LIN {X 0,Y 114.701,Z 386.692,A -85,B 0,C 180,E1 -25992.159,E2 -25992.159} C_VEL
LIN {X 0,Y 112.816,Z 386.681,A -85,B 0,C 180,E1 -25999.228,E2 -25999.228} C_VEL
LIN {X 0,Y 112.467,Z 385.169,A -85,B 0,C 180,E1 -26006.417,E2 -26006.417} C_VEL
LIN {X 0,Y 112.641,Z 383.781,A -85,B 0,C 180,E1 -26009.999,E2 -26009.999} C_VEL
LIN {X 0,Y 112.455,Z 380.804,A -85,B 0,C 180,E1 -26015.378,E2 -26015.378} C_VEL
LIN {X 0,Y 112.837,Z 376.72,A -85,B 0,C 180,E1 -26020.769,E2 -26020.769} C_VEL
LIN {X 0,Y 114.222,Z 370.392,A -85,B 0,C 180,E1 -26026.993,E2 -26026.993} C_VEL
LIN {X 0,Y 116.442,Z 363.485,A -85,B 0,C 180,E1 -26032.161,E2 -26032.161} C_VEL
LIN {X 0,Y 118.813,Z 356.389,A -85,B 0,C 180,E1 -26036.336,E2 -26036.336} C_VEL
LIN {X 0,Y 120.686,Z 351.028,A -85,B 0,C 180,E1 -26038.937,E2 -26038.937} C_VEL
LIN {X 0,Y 123.681,Z 342.854,A -85,B 0,C 180,E1 -26042.189,E2 -26042.189} C_VEL
LIN {X 0,Y 127.076,Z 332.271,A -85,B 0,C 180,E1 -26045.5,E2 -26045.5} C_VEL
LIN {X 0,Y 129.058,Z 325.849,A -85,B 0,C 180,E1 -26047.105,E2 -26047.105} C_VEL
LIN {X 0,Y 129.821,Z 322.45,A -85,B 0,C 180,E1 -26047.931,E2 -26047.931} C_VEL
LIN {X 0,Y 129.907,Z 315.621,A -85,B 0,C 180,E1 -26049.725,E2 -26049.725} C_VEL
LIN {X 0,Y 129.031,Z 304.225,A -85,B 0,C 180,E1 -26052.426,E2 -26052.426} C_VEL
LIN {X 0,Y 129.487,Z 298.65,A -85,B 0,C 180,E1 -26053.261,E2 -26053.261} C_VEL
LIN {X 0,Y 129.674,Z 297.694,A -85,B 0,C 180,E1 -26053.354,E2 -26053.354} C_VEL
LIN {X 0,Y 131.69,Z 283.784,A -85,B 0,C 180,E1 -26054.55,E2 -26054.55} C_VEL
LIN {X 0,Y 134.432,Z 245.397,A -85,B 0,C 180,E1 -26056.42,E2 -26056.42} C_VEL
LIN {X 0,Y 133.527,Z 229.449,A -85,B 0,C 180,E1 -26057.848,E2 -26057.848} C_VEL
LIN {X 0,Y 129.833,Z 218.225,A -85,B 0,C 180,E1 -26060.042,E2 -26060.042} C_VEL
LIN {X 0,Y 125.815,Z 208.24,A -85,B 0,C 180,E1 -26062.464,E2 -26062.464} C_VEL
LIN {X 0,Y 123.844,Z 204.228,A -85,B 0,C 180,E1 -26063.668,E2 -26063.668} C_VEL
LIN {X 0,Y 119.247,Z 196.971,A -85,B 0,C 180,E1 -26066.553,E2 -26066.553} C_VEL
LIN {X 0,Y 116.624,Z 193.11,A -85,B 0,C 180,E1 -26068.355,E2 -26068.355} C_VEL
LIN {X 0,Y 114.457,Z 189.787,A -85,B 0,C 180,E1 -26069.974,E2 -26069.974} C_VEL
LIN {X 0,Y 112.098,Z 186.672,A -85,B 0,C 180,E1 -26071.824,E2 -26071.824} C_VEL
LIN {X 0,Y 111.318,Z 185.287,A -85,B 0,C 180,E1 -26072.504,E2 -26072.504} C_VEL
LIN {X 0,Y 109.012,Z 183.185,A -85,B 0,C 180,E1 -26074.399,E2 -26074.399} C_VEL
LIN {X 0,Y 107.991,Z 180.792,A -85,B 0,C 180,E1 -26075.47,E2 -26075.47} C_VEL
LIN {X 0,Y 107.875,Z 180.047,A -85,B 0,C 180,E1 -26075.795,E2 -26075.795} C_VEL
LIN {X 0,Y 107.882,Z 179.983,A -85,B 0,C 180,E1 -26080.99,E2 -26080.99} C_VEL
LIN {X 0,Y 108.226,Z 180,A -85,B 0,C 180,E1 -26088.765,E2 -26088.765} C_VEL
LIN {X 0,Y 108.441,Z 179.966,A -85,B 0,C 180,E1 -26096.283,E2 -26096.283} C_VEL
LIN {X 0,Y 108.917,Z 179.902,A -85,B 0,C 180,E1 -26099.999,E2 -26099.999} C_VEL
LIN {X 0,Y 108.304,Z 179.989,A -85,B 0,C 180,E1 -26107.456,E2 -26107.456} C_VEL
LIN {X 0,Y 108.174,Z 179.988,A -85,B 0,C 180,E1 -26112.96,E2 -26112.96} C_VEL
LIN {X 0,Y 107.903,Z 180.028,A -85,B 0,C 180,E1 -26119.005,E2 -26119.005} C_VEL
LIN {X 0,Y 107.855,Z 180.044,A -85,B 0,C 180,E1 -26124.182,E2 -26124.182} C_VEL
LIN {X 0,Y 107.778,Z 180.041,A -85,B 0,C 180,E1 -26132.039,E2 -26132.039} C_VEL
LIN {X 0,Y 107.688,Z 180.049,A -85,B 0,C 180,E1 -26138.451,E2 -26138.451} C_VEL
LIN {X 0,Y 107.687,Z 180.208,A -85,B 0,C 180,E1 -26144.963,E2 -26144.963} C_VEL
LIN {X 0,Y 108.581,Z 182.753,A -85,B 0,C 180,E1 -26145.968,E2 -26145.968} C_VEL
LIN {X 0,Y 110.766,Z 185.022,A -85,B 0,C 180,E1 -26147.829,E2 -26147.829} C_VEL
LIN {X 0,Y 111.609,Z 185.761,A -85,B 0,C 180,E1 -26148.498,E2 -26148.498} C_VEL
LIN {X 0,Y 113.569,Z 188.992,A -85,B 0,C 180,E1 -26150.138,E2 -26150.138} C_VEL
LIN {X 0,Y 115.129,Z 190.684,A -85,B 0,C 180,E1 -26151.28,E2 -26151.28} C_VEL
LIN {X 0,Y 120.859,Z 199.285,A -85,B 0,C 180,E1 -26155.238,E2 -26155.238} C_VEL
LIN {X 0,Y 125.031,Z 206.174,A -85,B 0,C 180,E1 -26157.785,E2 -26157.785} C_VEL
LIN {X 0,Y 130.851,Z 217.027,A -85,B 0,C 180,E1 -26161.01,E2 -26161.01} C_VEL
LIN {X 0,Y 135.488,Z 227.713,A -85,B 0,C 180,E1 -26163.46,E2 -26163.46} C_VEL
LIN {X 0,Y 132.145,Z 273.455,A -85,B 0,C 180,E1 -26165.609,E2 -26165.609} C_VEL
LIN {X 0,Y 130.472,Z 286.832,A -85,B 0,C 180,E1 -26166.792,E2 -26166.792} C_VEL
LIN {X 0,Y 128.112,Z 299.797,A -85,B 0,C 180,E1 -26168.525,E2 -26168.525} C_VEL
LIN {X 0,Y 125.177,Z 311.686,A -85,B 0,C 180,E1 -26170.741,E2 -26170.741} C_VEL
LIN {X 0,Y 121.73,Z 323.3,A -85,B 0,C 180,E1 -26173.654,E2 -26173.654} C_VEL
LIN {X 0,Y 118.203,Z 333.75,A -85,B 0,C 180,E1 -26177.118,E2 -26177.118} C_VEL
LIN {X 0,Y 114.672,Z 343.135,A -85,B 0,C 180,E1 -26181.187,E2 -26181.187} C_VEL
LIN {X 0,Y 111.181,Z 352.262,A -85,B 0,C 180,E1 -26186.376,E2 -26186.376} C_VEL
LIN {X 0,Y 108.53,Z 359.552,A -85,B 0,C 180,E1 -26191.856,E2 -26191.856} C_VEL
LIN {X 0,Y 106.453,Z 365.739,A -85,B 0,C 180,E1 -26197.993,E2 -26197.993} C_VEL
LIN {X 0,Y 105.375,Z 369.965,A -85,B 0,C 180,E1 -26203.5,E2 -26203.5} C_VEL
LIN {X 0,Y 104.938,Z 373.8,A -85,B 0,C 180,E1 -26210.347,E2 -26210.347} C_VEL
LIN {X 0,Y 105.788,Z 376.41,A -85,B 0,C 180,E1 -26217.714,E2 -26217.714} C_VEL
LIN {X 0,Y 106.874,Z 377.199,A -85,B 0,C 180,E1 -26221.742,E2 -26221.742} C_VEL
LIN {X 0,Y 108.366,Z 377.569,A -85,B 0,C 180,E1 -26225.711,E2 -26225.711} C_VEL
LIN {X 0,Y 110.875,Z 377.373,A -85,B 0,C 180,E1 -26230.48,E2 -26230.48} C_VEL
LIN {X 0,Y 115.497,Z 375.922,A -85,B 0,C 180,E1 -26236.904,E2 -26236.904} C_VEL
LIN {X 0,Y 118.712,Z 374.445,A -85,B 0,C 180,E1 -26240.321,E2 -26240.321} C_VEL
LIN {X 0,Y 125.327,Z 370.597,A -85,B 0,C 180,E1 -26245.891,E2 -26245.891} C_VEL
LIN {X 0,Y 132.858,Z 365.177,A -85,B 0,C 180,E1 -26250.79,E2 -26250.79} C_VEL
LIN {X 0,Y 140.026,Z 358.919,A -85,B 0,C 180,E1 -26254.614,E2 -26254.614} C_VEL
LIN {X 0,Y 147.752,Z 351.022,A -85,B 0,C 180,E1 -26258.03,E2 -26258.03} C_VEL
LIN {X 0,Y 154.642,Z 342.793,A -85,B 0,C 180,E1 -26260.567,E2 -26260.567} C_VEL
LIN {X 0,Y 161.719,Z 332.547,A -85,B 0,C 180,E1 -26262.957,E2 -26262.957} C_VEL
LIN {X 0,Y 167.578,Z 322.406,A -85,B 0,C 180,E1 -26264.709,E2 -26264.709} C_VEL
LIN {X 0,Y 172.609,Z 311.679,A -85,B 0,C 180,E1 -26266.157,E2 -26266.157} C_VEL
LIN {X 0,Y 176.952,Z 300.005,A -85,B 0,C 180,E1 -26267.306,E2 -26267.306} C_VEL
LIN {X 0,Y 180.318,Z 287.878,A -85,B 0,C 180,E1 -26268.188,E2 -26268.188} C_VEL
LIN {X 0,Y 182.718,Z 275.29,A -85,B 0,C 180,E1 -26268.804,E2 -26268.804} C_VEL
LIN {X 0,Y 183.684,Z 266.817,A -85,B 0,C 180,E1 -26269.111,E2 -26269.111} C_VEL
LIN {X 0,Y 180.644,Z 260.298,A -85,B 0,C 180,E1 -26272.521,E2 -26272.521} C_VEL
LIN {X 0,Y 177.733,Z 254.302,A -85,B 0,C 180,E1 -26276.657,E2 -26276.657} C_VEL
LIN {X 0,Y 176.128,Z 251.308,A -85,B 0,C 180,E1 -26279.593,E2 -26279.593} C_VEL
LIN {X 0,Y 174.589,Z 248.05,A -85,B 0,C 180,E1 -26284.04,E2 -26284.04} C_VEL
LIN {X 0,Y 174.347,Z 247.326,A -85,B 0,C 180,E1 -26285.204,E2 -26285.204} C_VEL
LIN {X 0,Y 173.89,Z 247.213,A -85,B 0,C 180,E1 -26291.659,E2 -26291.659} C_VEL
LIN {X 0,Y 174.227,Z 247.599,A -85,B 0,C 180,E1 -26293.856,E2 -26293.856} C_VEL
LIN {X 0,Y 175.605,Z 251.412,A -85,B 0,C 180,E1 -26298.89,E2 -26298.89} C_VEL
LIN {X 0,Y 176.463,Z 253.601,A -85,B 0,C 180,E1 -26300.831,E2 -26300.831} C_VEL
LIN {X 0,Y 178.028,Z 257.372,A -85,B 0,C 180,E1 -26303.634,E2 -26303.634} C_VEL
LIN {X 0,Y 179.981,Z 262.71,A -85,B 0,C 180,E1 -26306.563,E2 -26306.563} C_VEL
LIN {X 0,Y 182.016,Z 268.722,A -85,B 0,C 180,E1 -26309.175,E2 -26309.175} C_VEL
LIN {X 0,Y 183.184,Z 272.321,A -85,B 0,C 180,E1 -26310.497,E2 -26310.497} C_VEL
LIN {X 0,Y 181.43,Z 286.139,A -85,B 0,C 180,E1 -26311.025,E2 -26311.025} C_VEL
LIN {X 0,Y 178.365,Z 299.021,A -85,B 0,C 180,E1 -26311.617,E2 -26311.617} C_VEL
LIN {X 0,Y 174.048,Z 312.047,A -85,B 0,C 180,E1 -26312.549,E2 -26312.549} C_VEL
LIN {X 0,Y 168.989,Z 323.707,A -85,B 0,C 180,E1 -26313.718,E2 -26313.718} C_VEL
LIN {X 0,Y 162.609,Z 335.397,A -85,B 0,C 180,E1 -26315.335,E2 -26315.335} C_VEL
LIN {X 0,Y 156.424,Z 344.847,A -85,B 0,C 180,E1 -26317.108,E2 -26317.108} C_VEL
LIN {X 0,Y 149.851,Z 353.495,A -85,B 0,C 180,E1 -26319.299,E2 -26319.299} C_VEL
LIN {X 0,Y 142.285,Z 361.956,A -85,B 0,C 180,E1 -26322.191,E2 -26322.191} C_VEL
LIN {X 0,Y 135.158,Z 368.785,A -85,B 0,C 180,E1 -26325.413,E2 -26325.413} C_VEL
LIN {X 0,Y 128.542,Z 374.292,A -85,B 0,C 180,E1 -26328.997,E2 -26328.997} C_VEL
LIN {X 0,Y 121.331,Z 379.649,A -85,B 0,C 180,E1 -26334.189,E2 -26334.189} C_VEL
LIN {X 0,Y 117.646,Z 381.979,A -85,B 0,C 180,E1 -26337.476,E2 -26337.476} C_VEL
LIN {X 0,Y 111.974,Z 384.967,A -85,B 0,C 180,E1 -26343.937,E2 -26343.937} C_VEL
LIN {X 0,Y 109.699,Z 385.885,A -85,B 0,C 180,E1 -26347.393,E2 -26347.393} C_VEL
LIN {X 0,Y 106.683,Z 386.525,A -85,B 0,C 180,E1 -26354.721,E2 -26354.721} C_VEL
LIN {X 0,Y 105.409,Z 385.676,A -85,B 0,C 180,E1 -26362.336,E2 -26362.336} C_VEL
LIN {X 0,Y 105.48,Z 383.981,A -85,B 0,C 180,E1 -26368.092,E2 -26368.092} C_VEL
LIN {X 0,Y 105.459,Z 382.498,A -85,B 0,C 180,E1 -26371.524,E2 -26371.524} C_VEL
LIN {X 0,Y 105.446,Z 378.874,A -85,B 0,C 180,E1 -26377.66,E2 -26377.66} C_VEL
LIN {X 0,Y 106.167,Z 374.293,A -85,B 0,C 180,E1 -26383.396,E2 -26383.396} C_VEL
LIN {X 0,Y 108.144,Z 367.298,A -85,B 0,C 180,E1 -26389.948,E2 -26389.948} C_VEL
LIN {X 0,Y 110.77,Z 359.68,A -85,B 0,C 180,E1 -26395.357,E2 -26395.357} C_VEL
LIN {X 0,Y 113.549,Z 351.859,A -85,B 0,C 180,E1 -26399.679,E2 -26399.679} C_VEL
LIN {X 0,Y 116.939,Z 343.453,A -85,B 0,C 180,E1 -26403.257,E2 -26403.257} C_VEL
LIN {X 0,Y 120.499,Z 333.091,A -85,B 0,C 180,E1 -26406.713,E2 -26406.713} C_VEL
LIN {X 0,Y 123.614,Z 323.202,A -85,B 0,C 180,E1 -26409.234,E2 -26409.234} C_VEL
LIN {X 0,Y 126.699,Z 311.658,A -85,B 0,C 180,E1 -26411.465,E2 -26411.465} C_VEL
LIN {X 0,Y 129.288,Z 300.08,A -85,B 0,C 180,E1 -26413.069,E2 -26413.069} C_VEL
LIN {X 0,Y 129.674,Z 297.694,A -85,B 0,C 180,E1 -26413.354,E2 -26413.354} C_VEL
LIN {X 0,Y 130.345,Z 292.966,A -85,B 0,C 180,E1 -26413.874,E2 -26413.874} C_VEL
LIN {X 0,Y 130.243,Z 290.151,A -85,B 0,C 180,E1 -26414.275,E2 -26414.275} C_VEL
LIN {X 0,Y 129.287,Z 282.732,A -85,B 0,C 180,E1 -26415.44,E2 -26415.44} C_VEL
LIN {X 0,Y 127.603,Z 273.348,A -85,B 0,C 180,E1 -26416.792,E2 -26416.792} C_VEL
LIN {X 0,Y 127.324,Z 267.511,A -85,B 0,C 180,E1 -26417.311,E2 -26417.311} C_VEL
LIN {X 0,Y 128.86,Z 244.337,A -85,B 0,C 180,E1 -26418.461,E2 -26418.461} C_VEL
LIN {X 0,Y 128.067,Z 231.4,A -85,B 0,C 180,E1 -26419.737,E2 -26419.737} C_VEL
LIN {X 0,Y 124.718,Z 220.97,A -85,B 0,C 180,E1 -26421.914,E2 -26421.914} C_VEL
LIN {X 0,Y 120.764,Z 211.039,A -85,B 0,C 180,E1 -26424.538,E2 -26424.538} C_VEL
LIN {X 0,Y 117.152,Z 204.663,A -85,B 0,C 180,E1 -26426.962,E2 -26426.962} C_VEL
LIN {X 0,Y 113.319,Z 198.721,A -85,B 0,C 180,E1 -26429.763,E2 -26429.763} C_VEL
LIN {X 0,Y 110.992,Z 195.236,A -85,B 0,C 180,E1 -26431.638,E2 -26431.638} C_VEL
LIN {X 0,Y 108.042,Z 191.063,A -85,B 0,C 180,E1 -26434.213,E2 -26434.213} C_VEL
LIN {X 0,Y 105.846,Z 188.492,A -85,B 0,C 180,E1 -26436.262,E2 -26436.262} C_VEL
LIN {X 0,Y 104.885,Z 186.451,A -85,B 0,C 180,E1 -26437.338,E2 -26437.338} C_VEL
LIN {X 0,Y 102.468,Z 184.637,A -85,B 0,C 180,E1 -26439.812,E2 -26439.812} C_VEL
LIN {X 0,Y 101.07,Z 182.025,A -85,B 0,C 180,E1 -26441.633,E2 -26441.633} C_VEL
LIN {X 0,Y 100.815,Z 180.859,A -85,B 0,C 180,E1 -26442.242,E2 -26442.242} C_VEL
LIN {X 0,Y 101.125,Z 180.879,A -85,B 0,C 180,E1 -26447.965,E2 -26447.965} C_VEL
LIN {X 0,Y 101.232,Z 180.856,A -85,B 0,C 180,E1 -26452.018,E2 -26452.018} C_VEL
LIN {X 0,Y 101.844,Z 180.782,A -85,B 0,C 180,E1 -26459.999,E2 -26459.999} C_VEL
LIN {X 0,Y 101.243,Z 180.866,A -85,B 0,C 180,E1 -26467.98,E2 -26467.98} C_VEL
LIN {X 0,Y 101.103,Z 180.87,A -85,B 0,C 180,E1 -26473.302,E2 -26473.302} C_VEL
LIN {X 0,Y 100.815,Z 180.902,A -85,B 0,C 180,E1 -26480.398,E2 -26480.398} C_VEL
LIN {X 0,Y 100.773,Z 180.93,A -85,B 0,C 180,E1 -26484.958,E2 -26484.958} C_VEL
LIN {X 0,Y 100.687,Z 180.932,A -85,B 0,C 180,E1 -26493.114,E2 -26493.114} C_VEL
LIN {X 0,Y 100.666,Z 180.974,A -85,B 0,C 180,E1 -26498.526,E2 -26498.526} C_VEL
LIN {X 0,Y 101.319,Z 183.24,A -85,B 0,C 180,E1 -26499.581,E2 -26499.581} C_VEL
LIN {X 0,Y 103.297,Z 185.672,A -85,B 0,C 180,E1 -26501.894,E2 -26501.894} C_VEL
LIN {X 0,Y 104.844,Z 186.814,A -85,B 0,C 180,E1 -26503.443,E2 -26503.443} C_VEL
LIN {X 0,Y 106.693,Z 189.893,A -85,B 0,C 180,E1 -26505.367,E2 -26505.367} C_VEL
LIN {X 0,Y 108.713,Z 192.013,A -85,B 0,C 180,E1 -26507.153,E2 -26507.153} C_VEL
LIN {X 0,Y 111.364,Z 195.716,A -85,B 0,C 180,E1 -26509.413,E2 -26509.413} C_VEL
LIN {X 0,Y 115.239,Z 201.557,A -85,B 0,C 180,E1 -26512.421,E2 -26512.421} C_VEL
LIN {X 0,Y 120.179,Z 209.544,A -85,B 0,C 180,E1 -26515.801,E2 -26515.801} C_VEL
LIN {X 0,Y 126.22,Z 221.191,A -85,B 0,C 180,E1 -26519.494,E2 -26519.494} C_VEL
LIN {X 0,Y 129.832,Z 229.561,A -85,B 0,C 180,E1 -26521.553,E2 -26521.553} C_VEL
LIN {X 0,Y 126.447,Z 274.354,A -85,B 0,C 180,E1 -26523.746,E2 -26523.746} C_VEL
LIN {X 0,Y 124.618,Z 287.912,A -85,B 0,C 180,E1 -26524.995,E2 -26524.995} C_VEL
LIN {X 0,Y 122.241,Z 300.262,A -85,B 0,C 180,E1 -26526.718,E2 -26526.718} C_VEL
LIN {X 0,Y 119.343,Z 311.486,A -85,B 0,C 180,E1 -26528.858,E2 -26528.858} C_VEL
LIN {X 0,Y 115.681,Z 323.201,A -85,B 0,C 180,E1 -26531.859,E2 -26531.859} C_VEL
LIN {X 0,Y 111.932,Z 333.741,A -85,B 0,C 180,E1 -26535.455,E2 -26535.455} C_VEL
LIN {X 0,Y 108.271,Z 343.007,A -85,B 0,C 180,E1 -26539.616,E2 -26539.616} C_VEL
LIN {X 0,Y 104.458,Z 352.362,A -85,B 0,C 180,E1 -26545.176,E2 -26545.176} C_VEL
LIN {X 0,Y 101.627,Z 359.708,A -85,B 0,C 180,E1 -26550.991,E2 -26550.991} C_VEL
LIN {X 0,Y 99.326,Z 366.195,A -85,B 0,C 180,E1 -26557.867,E2 -26557.867} C_VEL
LIN {X 0,Y 98.132,Z 370.85,A -85,B 0,C 180,E1 -26564.518,E2 -26564.518} C_VEL
LIN {X 0,Y 97.852,Z 374.164,A -85,B 0,C 180,E1 -26571.047,E2 -26571.047} C_VEL
LIN {X 0,Y 98.244,Z 375.791,A -85,B 0,C 180,E1 -26575.419,E2 -26575.419} C_VEL
LIN {X 0,Y 99.896,Z 377.43,A -85,B 0,C 180,E1 -26582.411,E2 -26582.411} C_VEL
LIN {X 0,Y 102.222,Z 377.932,A -85,B 0,C 180,E1 -26588.227,E2 -26588.227} C_VEL
LIN {X 0,Y 104.541,Z 377.719,A -85,B 0,C 180,E1 -26592.312,E2 -26592.312} C_VEL
LIN {X 0,Y 107.212,Z 377.092,A -85,B 0,C 180,E1 -26596.145,E2 -26596.145} C_VEL
LIN {X 0,Y 111.36,Z 375.573,A -85,B 0,C 180,E1 -26600.869,E2 -26600.869} C_VEL
LIN {X 0,Y 117.901,Z 372.339,A -85,B 0,C 180,E1 -26606.568,E2 -26606.568} C_VEL
LIN {X 0,Y 124.496,Z 368.233,A -85,B 0,C 180,E1 -26611.046,E2 -26611.046} C_VEL
LIN {X 0,Y 131.763,Z 362.775,A -85,B 0,C 180,E1 -26615.061,E2 -26615.061} C_VEL
LIN {X 0,Y 139.582,Z 355.769,A -85,B 0,C 180,E1 -26618.668,E2 -26618.668} C_VEL
LIN {X 0,Y 146.374,Z 348.696,A -85,B 0,C 180,E1 -26621.277,E2 -26621.277} C_VEL
LIN {X 0,Y 153.726,Z 339.698,A -85,B 0,C 180,E1 -26623.756,E2 -26623.756} C_VEL
LIN {X 0,Y 160.409,Z 329.813,A -85,B 0,C 180,E1 -26625.782,E2 -26625.782} C_VEL
LIN {X 0,Y 166.392,Z 319.026,A -85,B 0,C 180,E1 -26627.46,E2 -26627.46} C_VEL
LIN {X 0,Y 171.325,Z 308.107,A -85,B 0,C 180,E1 -26628.732,E2 -26628.732} C_VEL
LIN {X 0,Y 175.544,Z 296.066,A -85,B 0,C 180,E1 -26629.785,E2 -26629.785} C_VEL
LIN {X 0,Y 178.732,Z 283.464,A -85,B 0,C 180,E1 -26630.542,E2 -26630.542} C_VEL
LIN {X 0,Y 180.761,Z 270.84,A -85,B 0,C 180,E1 -26631.053,E2 -26631.053} C_VEL
LIN {X 0,Y 178.005,Z 264.538,A -85,B 0,C 180,E1 -26634.689,E2 -26634.689} C_VEL
LIN {X 0,Y 175.873,Z 260.138,A -85,B 0,C 180,E1 -26638.171,E2 -26638.171} C_VEL
LIN {X 0,Y 174.892,Z 258.049,A -85,B 0,C 180,E1 -26640.253,E2 -26640.253} C_VEL
LIN {X 0,Y 173.536,Z 254.812,A -85,B 0,C 180,E1 -26644.646,E2 -26644.646} C_VEL
LIN {X 0,Y 173.3,Z 254.338,A -85,B 0,C 180,E1 -26645.819,E2 -26645.819} C_VEL
LIN {X 0,Y 172.996,Z 254.247,A -85,B 0,C 180,E1 -26651.72,E2 -26651.72} C_VEL
LIN {X 0,Y 173.246,Z 254.591,A -85,B 0,C 180,E1 -26653.481,E2 -26653.481} C_VEL
LIN {X 0,Y 174.536,Z 258.424,A -85,B 0,C 180,E1 -26658.572,E2 -26658.572} C_VEL
LIN {X 0,Y 176.437,Z 263.611,A -85,B 0,C 180,E1 -26662.66,E2 -26662.66} C_VEL
LIN {X 0,Y 178.367,Z 269.331,A -85,B 0,C 180,E1 -26665.819,E2 -26665.819} C_VEL
LIN {X 0,Y 180.311,Z 275.713,A -85,B 0,C 180,E1 -26668.541,E2 -26668.541} C_VEL
LIN {X 0,Y 178.03,Z 289.665,A -85,B 0,C 180,E1 -26669.063,E2 -26669.063} C_VEL
LIN {X 0,Y 174.813,Z 301.773,A -85,B 0,C 180,E1 -26669.672,E2 -26669.672} C_VEL
LIN {X 0,Y 170.378,Z 313.955,A -85,B 0,C 180,E1 -26670.561,E2 -26670.561} C_VEL
LIN {X 0,Y 165.187,Z 325.092,A -85,B 0,C 180,E1 -26671.688,E2 -26671.688} C_VEL
LIN {X 0,Y 158.639,Z 336.483,A -85,B 0,C 180,E1 -26673.259,E2 -26673.259} C_VEL
LIN {X 0,Y 152.276,Z 345.689,A -85,B 0,C 180,E1 -26674.993,E2 -26674.993} C_VEL
LIN {X 0,Y 144.142,Z 355.597,A -85,B 0,C 180,E1 -26677.597,E2 -26677.597} C_VEL
LIN {X 0,Y 136.371,Z 363.605,A -85,B 0,C 180,E1 -26680.522,E2 -26680.522} C_VEL
LIN {X 0,Y 130.207,Z 369.07,A -85,B 0,C 180,E1 -26683.224,E2 -26683.224} C_VEL
LIN {X 0,Y 123.284,Z 374.455,A -85,B 0,C 180,E1 -26686.836,E2 -26686.836} C_VEL
LIN {X 0,Y 117.128,Z 378.697,A -85,B 0,C 180,E1 -26690.947,E2 -26690.947} C_VEL
LIN {X 0,Y 111.704,Z 381.924,A -85,B 0,C 180,E1 -26695.51,E2 -26695.51} C_VEL
LIN {X 0,Y 105.618,Z 384.809,A -85,B 0,C 180,E1 -26702.238,E2 -26702.238} C_VEL
LIN {X 0,Y 101.203,Z 386.087,A -85,B 0,C 180,E1 -26709.682,E2 -26709.682} C_VEL
LIN {X 0,Y 98.863,Z 385.891,A -85,B 0,C 180,E1 -26717.685,E2 -26717.685} C_VEL
LIN {X 0,Y 98.355,Z 385.224,A -85,B 0,C 180,E1 -26721.783,E2 -26721.783} C_VEL
LIN {X 0,Y 98.431,Z 383.287,A -85,B 0,C 180,E1 -26728.416,E2 -26728.416} C_VEL
LIN {X 0,Y 98.31,Z 380.639,A -85,B 0,C 180,E1 -26734.099,E2 -26734.099} C_VEL
LIN {X 0,Y 98.572,Z 376.721,A -85,B 0,C 180,E1 -26740.267,E2 -26740.267} C_VEL
LIN {X 0,Y 99.993,Z 370.632,A -85,B 0,C 180,E1 -26747.379,E2 -26747.379} C_VEL
LIN {X 0,Y 102.36,Z 363.924,A -85,B 0,C 180,E1 -26753.252,E2 -26753.252} C_VEL
LIN {X 0,Y 105.496,Z 355.533,A -85,B 0,C 180,E1 -26758.88,E2 -26758.88} C_VEL
LIN {X 0,Y 108.199,Z 348.95,A -85,B 0,C 180,E1 -26762.293,E2 -26762.293} C_VEL
LIN {X 0,Y 111.777,Z 339.734,A -85,B 0,C 180,E1 -26766.118,E2 -26766.118} C_VEL
LIN {X 0,Y 114.775,Z 331.263,A -85,B 0,C 180,E1 -26768.875,E2 -26768.875} C_VEL
LIN {X 0,Y 118.643,Z 319.446,A -85,B 0,C 180,E1 -26771.79,E2 -26771.79} C_VEL
LIN {X 0,Y 121.992,Z 306.784,A -85,B 0,C 180,E1 -26774.02,E2 -26774.02} C_VEL
LIN {X 0,Y 124.677,Z 293.418,A -85,B 0,C 180,E1 -26775.658,E2 -26775.658} C_VEL
LIN {X 0,Y 126.416,Z 280.076,A -85,B 0,C 180,E1 -26776.667,E2 -26776.667} C_VEL
LIN {X 0,Y 127.324,Z 267.511,A -85,B 0,C 180,E1 -26777.311,E2 -26777.311} C_VEL
LIN {X 0,Y 127.146,Z 261.686,A -85,B 0,C 180,E1 -26777.809,E2 -26777.809} C_VEL
LIN {X 0,Y 125.583,Z 252.305,A -85,B 0,C 180,E1 -26779.114,E2 -26779.114} C_VEL
LIN {X 0,Y 123.455,Z 241.084,A -85,B 0,C 180,E1 -26780.84,E2 -26780.84} C_VEL
LIN {X 0,Y 123.097,Z 237.226,A -85,B 0,C 180,E1 -26781.299,E2 -26781.299} C_VEL
LIN {X 0,Y 122.759,Z 233.368,A -85,B 0,C 180,E1 -26781.755,E2 -26781.755} C_VEL
LIN {X 0,Y 119.133,Z 222.078,A -85,B 0,C 180,E1 -26784.369,E2 -26784.369} C_VEL
LIN {X 0,Y 115.868,Z 214.01,A -85,B 0,C 180,E1 -26786.783,E2 -26786.783} C_VEL
LIN {X 0,Y 110.547,Z 204.935,A -85,B 0,C 180,E1 -26790.885,E2 -26790.885} C_VEL
LIN {X 0,Y 107.505,Z 200.444,A -85,B 0,C 180,E1 -26793.524,E2 -26793.524} C_VEL
LIN {X 0,Y 105.228,Z 197.043,A -85,B 0,C 180,E1 -26795.688,E2 -26795.688} C_VEL
LIN {X 0,Y 102.784,Z 193.818,A -85,B 0,C 180,E1 -26798.216,E2 -26798.216} C_VEL
LIN {X 0,Y 102.037,Z 192.616,A -85,B 0,C 180,E1 -26799.083,E2 -26799.083} C_VEL
LIN {X 0,Y 99.562,Z 190.02,A -85,B 0,C 180,E1 -26802.011,E2 -26802.011} C_VEL
LIN {X 0,Y 98.284,Z 187.472,A -85,B 0,C 180,E1 -26803.913,E2 -26803.913} C_VEL
LIN {X 0,Y 95.817,Z 185.626,A -85,B 0,C 180,E1 -26807.557,E2 -26807.557} C_VEL
LIN {X 0,Y 94.45,Z 183.265,A -85,B 0,C 180,E1 -26810.226,E2 -26810.226} C_VEL
LIN {X 0,Y 94.14,Z 181.743,A -85,B 0,C 180,E1 -26811.277,E2 -26811.277} C_VEL
LIN {X 0,Y 94.773,Z 181.661,A -85,B 0,C 180,E1 -26819.999,E2 -26819.999} C_VEL
LIN {X 0,Y 94.176,Z 181.741,A -85,B 0,C 180,E1 -26828.583,E2 -26828.583} C_VEL
LIN {X 0,Y 94.023,Z 181.753,A -85,B 0,C 180,E1 -26833.662,E2 -26833.662} C_VEL
LIN {X 0,Y 93.69,Z 181.789,A -85,B 0,C 180,E1 -26842.027,E2 -26842.027} C_VEL
LIN {X 0,Y 93.629,Z 181.964,A -85,B 0,C 180,E1 -26848.741,E2 -26848.741} C_VEL
LIN {X 0,Y 94.38,Z 184.288,A -85,B 0,C 180,E1 -26850.637,E2 -26850.637} C_VEL
LIN {X 0,Y 96.689,Z 186.837,A -85,B 0,C 180,E1 -26854.673,E2 -26854.673} C_VEL
LIN {X 0,Y 98.31,Z 187.833,A -85,B 0,C 180,E1 -26856.937,E2 -26856.937} C_VEL
LIN {X 0,Y 99.925,Z 190.819,A -85,B 0,C 180,E1 -26859.27,E2 -26859.27} C_VEL
LIN {X 0,Y 102.339,Z 193.289,A -85,B 0,C 180,E1 -26862.061,E2 -26862.061} C_VEL
LIN {X 0,Y 104.697,Z 196.675,A -85,B 0,C 180,E1 -26864.594,E2 -26864.594} C_VEL
LIN {X 0,Y 105.935,Z 198.189,A -85,B 0,C 180,E1 -26865.783,E2 -26865.783} C_VEL
LIN {X 0,Y 110.851,Z 205.318,A -85,B 0,C 180,E1 -26870.103,E2 -26870.103} C_VEL
LIN {X 0,Y 116.343,Z 214.711,A -85,B 0,C 180,E1 -26874.292,E2 -26874.292} C_VEL
LIN {X 0,Y 121.605,Z 225.166,A -85,B 0,C 180,E1 -26877.816,E2 -26877.816} C_VEL
LIN {X 0,Y 124.353,Z 231.71,A -85,B 0,C 180,E1 -26879.549,E2 -26879.549} C_VEL
LIN {X 0,Y 120.907,Z 274.78,A -85,B 0,C 180,E1 -26881.694,E2 -26881.694} C_VEL
LIN {X 0,Y 118.916,Z 288.704,A -85,B 0,C 180,E1 -26883.016,E2 -26883.016} C_VEL
LIN {X 0,Y 116.547,Z 300.366,A -85,B 0,C 180,E1 -26884.692,E2 -26884.692} C_VEL
LIN {X 0,Y 113.159,Z 312.786,A -85,B 0,C 180,E1 -26887.16,E2 -26887.16} C_VEL
LIN {X 0,Y 109.304,Z 324.329,A -85,B 0,C 180,E1 -26890.272,E2 -26890.272} C_VEL
LIN {X 0,Y 105.357,Z 334.692,A -85,B 0,C 180,E1 -26894.029,E2 -26894.029} C_VEL
LIN {X 0,Y 101.232,Z 344.444,A -85,B 0,C 180,E1 -26898.741,E2 -26898.741} C_VEL
LIN {X 0,Y 97.791,Z 352.412,A -85,B 0,C 180,E1 -26903.812,E2 -26903.812} C_VEL
LIN {X 0,Y 94.733,Z 359.824,A -85,B 0,C 180,E1 -26910.001,E2 -26910.001} C_VEL
LIN {X 0,Y 92.215,Z 366.673,A -85,B 0,C 180,E1 -26917.796,E2 -26917.796} C_VEL
LIN {X 0,Y 90.916,Z 371.708,A -85,B 0,C 180,E1 -26925.698,E2 -26925.698} C_VEL
LIN {X 0,Y 90.84,Z 374.877,A -85,B 0,C 180,E1 -26932.759,E2 -26932.759} C_VEL
LIN {X 0,Y 91.449,Z 376.376,A -85,B 0,C 180,E1 -26937.46,E2 -26937.46} C_VEL
LIN {X 0,Y 93.188,Z 377.756,A -85,B 0,C 180,E1 -26943.944,E2 -26943.944} C_VEL
LIN {X 0,Y 96.315,Z 378.245,A -85,B 0,C 180,E1 -26951.051,E2 -26951.051} C_VEL
LIN {X 0,Y 98.939,Z 377.97,A -85,B 0,C 180,E1 -26955.264,E2 -26955.264} C_VEL
LIN {X 0,Y 102.008,Z 377.26,A -85,B 0,C 180,E1 -26959.277,E2 -26959.277} C_VEL
LIN {X 0,Y 105.832,Z 375.929,A -85,B 0,C 180,E1 -26963.298,E2 -26963.298} C_VEL
LIN {X 0,Y 111.62,Z 373.33,A -85,B 0,C 180,E1 -26968.214,E2 -26968.214} C_VEL
LIN {X 0,Y 118.513,Z 369.456,A -85,B 0,C 180,E1 -26972.815,E2 -26972.815} C_VEL
LIN {X 0,Y 126.458,Z 364.003,A -85,B 0,C 180,E1 -26977.106,E2 -26977.106} C_VEL
LIN {X 0,Y 134.166,Z 357.654,A -85,B 0,C 180,E1 -26980.545,E2 -26980.545} C_VEL
LIN {X 0,Y 141.314,Z 350.755,A -85,B 0,C 180,E1 -26983.211,E2 -26983.211} C_VEL
LIN {X 0,Y 148.735,Z 342.318,A -85,B 0,C 180,E1 -26985.62,E2 -26985.62} C_VEL
LIN {X 0,Y 156.379,Z 331.889,A -85,B 0,C 180,E1 -26987.819,E2 -26987.819} C_VEL
LIN {X 0,Y 162.631,Z 321.42,A -85,B 0,C 180,E1 -26989.463,E2 -26989.463} C_VEL
LIN {X 0,Y 167.361,Z 311.76,A -85,B 0,C 180,E1 -26990.628,E2 -26990.628} C_VEL
LIN {X 0,Y 172.241,Z 299.064,A -85,B 0,C 180,E1 -26991.776,E2 -26991.776} C_VEL
LIN {X 0,Y 175.875,Z 286.234,A -85,B 0,C 180,E1 -26992.579,E2 -26992.579} C_VEL
LIN {X 0,Y 177.946,Z 274.935,A -85,B 0,C 180,E1 -26993.125,E2 -26993.125} C_VEL
LIN {X 0,Y 176.043,Z 270.255,A -85,B 0,C 180,E1 -26996.123,E2 -26996.123} C_VEL
LIN {X 0,Y 174.602,Z 266.886,A -85,B 0,C 180,E1 -26998.761,E2 -26998.761} C_VEL
LIN {X 0,Y 173.699,Z 264.832,A -85,B 0,C 180,E1 -27000.87,E2 -27000.87} C_VEL
LIN {X 0,Y 172.504,Z 261.565,A -85,B 0,C 180,E1 -27005.26,E2 -27005.26} C_VEL
LIN {X 0,Y 171.975,Z 261.15,A -85,B 0,C 180,E1 -27009.409,E2 -27009.409} C_VEL
LIN {X 0,Y 172.265,Z 261.487,A -85,B 0,C 180,E1 -27013.004,E2 -27013.004} C_VEL
LIN {X 0,Y 173.388,Z 265.214,A -85,B 0,C 180,E1 -27018.004,E2 -27018.004} C_VEL
LIN {X 0,Y 174.927,Z 269.899,A -85,B 0,C 180,E1 -27021.72,E2 -27021.72} C_VEL
LIN {X 0,Y 176.66,Z 275.696,A -85,B 0,C 180,E1 -27024.917,E2 -27024.917} C_VEL
LIN {X 0,Y 177.555,Z 279.236,A -85,B 0,C 180,E1 -27026.465,E2 -27026.465} C_VEL
LIN {X 0,Y 174.957,Z 292.646,A -85,B 0,C 180,E1 -27027.021,E2 -27027.021} C_VEL
LIN {X 0,Y 171.443,Z 304.417,A -85,B 0,C 180,E1 -27027.64,E2 -27027.64} C_VEL
LIN {X 0,Y 166.919,Z 315.862,A -85,B 0,C 180,E1 -27028.486,E2 -27028.486} C_VEL
LIN {X 0,Y 161.607,Z 326.556,A -85,B 0,C 180,E1 -27029.568,E2 -27029.568} C_VEL
LIN {X 0,Y 154.888,Z 337.537,A -85,B 0,C 180,E1 -27031.079,E2 -27031.079} C_VEL
LIN {X 0,Y 148.346,Z 346.466,A -85,B 0,C 180,E1 -27032.762,E2 -27032.762} C_VEL
LIN {X 0,Y 141.345,Z 354.685,A -85,B 0,C 180,E1 -27034.872,E2 -27034.872} C_VEL
LIN {X 0,Y 133.188,Z 362.795,A -85,B 0,C 180,E1 -27037.672,E2 -27037.672} C_VEL
LIN {X 0,Y 125.454,Z 369.356,A -85,B 0,C 180,E1 -27040.862,E2 -27040.862} C_VEL
LIN {X 0,Y 118.203,Z 374.62,A -85,B 0,C 180,E1 -27044.48,E2 -27044.48} C_VEL
LIN {X 0,Y 111.697,Z 378.749,A -85,B 0,C 180,E1 -27048.649,E2 -27048.649} C_VEL
LIN {X 0,Y 105.899,Z 381.87,A -85,B 0,C 180,E1 -27053.323,E2 -27053.323} C_VEL
LIN {X 0,Y 102.424,Z 383.455,A -85,B 0,C 180,E1 -27056.705,E2 -27056.705} C_VEL
LIN {X 0,Y 96.732,Z 385.385,A -85,B 0,C 180,E1 -27064.155,E2 -27064.155} C_VEL
LIN {X 0,Y 92.98,Z 385.823,A -85,B 0,C 180,E1 -27072.401,E2 -27072.401} C_VEL
LIN {X 0,Y 91.932,Z 385.486,A -85,B 0,C 180,E1 -27076.741,E2 -27076.741} C_VEL
LIN {X 0,Y 91.234,Z 383.591,A -85,B 0,C 180,E1 -27085.581,E2 -27085.581} C_VEL
LIN {X 0,Y 91.368,Z 381.862,A -85,B 0,C 180,E1 -27090.445,E2 -27090.445} C_VEL
LIN {X 0,Y 91.235,Z 378.756,A -85,B 0,C 180,E1 -27096.634,E2 -27096.634} C_VEL
LIN {X 0,Y 91.887,Z 374.346,A -85,B 0,C 180,E1 -27103.264,E2 -27103.264} C_VEL
LIN {X 0,Y 93.545,Z 368.691,A -85,B 0,C 180,E1 -27109.759,E2 -27109.759} C_VEL
LIN {X 0,Y 96.333,Z 361.594,A -85,B 0,C 180,E1 -27115.958,E2 -27115.958} C_VEL
LIN {X 0,Y 99.753,Z 352.974,A -85,B 0,C 180,E1 -27121.645,E2 -27121.645} C_VEL
LIN {X 0,Y 103.928,Z 343.712,A -85,B 0,C 180,E1 -27126.157,E2 -27126.157} C_VEL
LIN {X 0,Y 107.939,Z 333.364,A -85,B 0,C 180,E1 -27130.013,E2 -27130.013} C_VEL
LIN {X 0,Y 110.819,Z 325.152,A -85,B 0,C 180,E1 -27132.362,E2 -27132.362} C_VEL
LIN {X 0,Y 114.48,Z 313.417,A -85,B 0,C 180,E1 -27134.909,E2 -27134.909} C_VEL
LIN {X 0,Y 117.552,Z 301.257,A -85,B 0,C 180,E1 -27136.772,E2 -27136.772} C_VEL
LIN {X 0,Y 119.951,Z 288.013,A -85,B 0,C 180,E1 -27138.175,E2 -27138.175} C_VEL
LIN {X 0,Y 121.339,Z 274.65,A -85,B 0,C 180,E1 -27139.04,E2 -27139.04} C_VEL
LIN {X 0,Y 123.467,Z 245.574,A -85,B 0,C 180,E1 -27140.478,E2 -27140.478} C_VEL
LIN {X 0,Y 123.097,Z 237.226,A -85,B 0,C 180,E1 -27141.299,E2 -27141.299} C_VEL
LIN {X 0,Y 122.378,Z 234.326,A -85,B 0,C 180,E1 -27141.842,E2 -27141.842} C_VEL
LIN {X 0,Y 120.244,Z 231.136,A -85,B 0,C 180,E1 -27143.062,E2 -27143.062} C_VEL
LIN {X 0,Y 115.059,Z 225.786,A -85,B 0,C 180,E1 -27146.116,E2 -27146.116} C_VEL
LIN {X 0,Y 113.525,Z 222.694,A -85,B 0,C 180,E1 -27147.255,E2 -27147.255} C_VEL
LIN {X 0,Y 111.305,Z 217.483,A -85,B 0,C 180,E1 -27149.084,E2 -27149.084} C_VEL
LIN {X 0,Y 106.393,Z 209.105,A -85,B 0,C 180,E1 -27153.333,E2 -27153.333} C_VEL
LIN {X 0,Y 102.606,Z 203.144,A -85,B 0,C 180,E1 -27157.113,E2 -27157.113} C_VEL
LIN {X 0,Y 99.918,Z 199.287,A -85,B 0,C 180,E1 -27160.197,E2 -27160.197} C_VEL
LIN {X 0,Y 97.015,Z 195.685,A -85,B 0,C 180,E1 -27164.034,E2 -27164.034} C_VEL
LIN {X 0,Y 96.15,Z 194.011,A -85,B 0,C 180,E1 -27165.447,E2 -27165.447} C_VEL
LIN {X 0,Y 93.742,Z 191.687,A -85,B 0,C 180,E1 -27169.501,E2 -27169.501} C_VEL
LIN {X 0,Y 92.432,Z 188.946,A -85,B 0,C 180,E1 -27172.528,E2 -27172.528} C_VEL
LIN {X 0,Y 91.916,Z 188.469,A -85,B 0,C 180,E1 -27173.713,E2 -27173.713} C_VEL
LIN {X 0,Y 89.507,Z 186.651,A -85,B 0,C 180,E1 -27181.124,E2 -27181.124} C_VEL
LIN {X 0,Y 88.495,Z 186.033,A -85,B 0,C 180,E1 -27189.138,E2 -27189.138} C_VEL
LIN {X 0,Y 88.794,Z 186.793,A -85,B 0,C 180,E1 -27196.082,E2 -27196.082} C_VEL
LIN {X 0,Y 91.923,Z 188.813,A -85,B 0,C 180,E1 -27207.181,E2 -27207.181} C_VEL
LIN {X 0,Y 93.183,Z 191.602,A -85,B 0,C 180,E1 -27210.289,E2 -27210.289} C_VEL
LIN {X 0,Y 95.906,Z 194.09,A -85,B 0,C 180,E1 -27214.988,E2 -27214.988} C_VEL
LIN {X 0,Y 98.723,Z 198.262,A -85,B 0,C 180,E1 -27219.136,E2 -27219.136} C_VEL
LIN {X 0,Y 99.974,Z 199.681,A -85,B 0,C 180,E1 -27220.675,E2 -27220.675} C_VEL
LIN {X 0,Y 103.383,Z 204.572,A -85,B 0,C 180,E1 -27224.506,E2 -27224.506} C_VEL
LIN {X 0,Y 107.495,Z 210.71,A -85,B 0,C 180,E1 -27228.41,E2 -27228.41} C_VEL
LIN {X 0,Y 112.299,Z 219.243,A -85,B 0,C 180,E1 -27232.444,E2 -27232.444} C_VEL
LIN {X 0,Y 117.25,Z 229.553,A -85,B 0,C 180,E1 -27236.117,E2 -27236.117} C_VEL
LIN {X 0,Y 119.073,Z 233.952,A -85,B 0,C 180,E1 -27237.389,E2 -27237.389} C_VEL
LIN {X 0,Y 115.572,Z 275.017,A -85,B 0,C 180,E1 -27239.444,E2 -27239.444} C_VEL
LIN {X 0,Y 113.487,Z 288.813,A -85,B 0,C 180,E1 -27240.764,E2 -27240.764} C_VEL
LIN {X 0,Y 110.89,Z 300.9,A -85,B 0,C 180,E1 -27242.534,E2 -27242.534} C_VEL
LIN {X 0,Y 107.596,Z 312.463,A -85,B 0,C 180,E1 -27244.877,E2 -27244.877} C_VEL
LIN {X 0,Y 103.486,Z 324.132,A -85,B 0,C 180,E1 -27248.068,E2 -27248.068} C_VEL
LIN {X 0,Y 99.29,Z 334.613,A -85,B 0,C 180,E1 -27251.961,E2 -27251.961} C_VEL
LIN {X 0,Y 94.705,Z 344.851,A -85,B 0,C 180,E1 -27257.137,E2 -27257.137} C_VEL
LIN {X 0,Y 91.177,Z 352.46,A -85,B 0,C 180,E1 -27262.249,E2 -27262.249} C_VEL
LIN {X 0,Y 87.871,Z 359.93,A -85,B 0,C 180,E1 -27268.855,E2 -27268.855} C_VEL
LIN {X 0,Y 85.438,Z 366.056,A -85,B 0,C 180,E1 -27276.142,E2 -27276.142} C_VEL
LIN {X 0,Y 83.912,Z 371.25,A -85,B 0,C 180,E1 -27284.553,E2 -27284.553} C_VEL
LIN {X 0,Y 83.741,Z 374.796,A -85,B 0,C 180,E1 -27292.607,E2 -27292.607} C_VEL
LIN {X 0,Y 84.768,Z 376.964,A -85,B 0,C 180,E1 -27299.832,E2 -27299.832} C_VEL
LIN {X 0,Y 86.532,Z 378.08,A -85,B 0,C 180,E1 -27305.691,E2 -27305.691} C_VEL
LIN {X 0,Y 90.664,Z 378.559,A -85,B 0,C 180,E1 -27314.24,E2 -27314.24} C_VEL
LIN {X 0,Y 93.673,Z 378.213,A -85,B 0,C 180,E1 -27318.615,E2 -27318.615} C_VEL
LIN {X 0,Y 100.49,Z 376.291,A -85,B 0,C 180,E1 -27325.98,E2 -27325.98} C_VEL
LIN {X 0,Y 107.762,Z 373.215,A -85,B 0,C 180,E1 -27331.697,E2 -27331.697} C_VEL
LIN {X 0,Y 115.205,Z 369.19,A -85,B 0,C 180,E1 -27336.217,E2 -27336.217} C_VEL
LIN {X 0,Y 123.981,Z 363.315,A -85,B 0,C 180,E1 -27340.508,E2 -27340.508} C_VEL
LIN {X 0,Y 131.811,Z 356.976,A -85,B 0,C 180,E1 -27343.689,E2 -27343.689} C_VEL
LIN {X 0,Y 139.304,Z 349.879,A -85,B 0,C 180,E1 -27346.213,E2 -27346.213} C_VEL
LIN {X 0,Y 147.746,Z 340.356,A -85,B 0,C 180,E1 -27348.671,E2 -27348.671} C_VEL
LIN {X 0,Y 154.956,Z 330.373,A -85,B 0,C 180,E1 -27350.567,E2 -27350.567} C_VEL
LIN {X 0,Y 161.403,Z 319.411,A -85,B 0,C 180,E1 -27352.144,E2 -27352.144} C_VEL
LIN {X 0,Y 166.898,Z 307.829,A -85,B 0,C 180,E1 -27353.347,E2 -27353.347} C_VEL
LIN {X 0,Y 171.267,Z 295.646,A -85,B 0,C 180,E1 -27354.294,E2 -27354.294} C_VEL
LIN {X 0,Y 174.657,Z 282.393,A -85,B 0,C 180,E1 -27355.013,E2 -27355.013} C_VEL
LIN {X 0,Y 175.246,Z 279.139,A -85,B 0,C 180,E1 -27355.184,E2 -27355.184} C_VEL
LIN {X 0,Y 173.324,Z 273.704,A -85,B 0,C 180,E1 -27359.274,E2 -27359.274} C_VEL
LIN {X 0,Y 172.529,Z 271.624,A -85,B 0,C 180,E1 -27361.459,E2 -27361.459} C_VEL
LIN {X 0,Y 171.477,Z 268.44,A -85,B 0,C 180,E1 -27365.881,E2 -27365.881} C_VEL
LIN {X 0,Y 171.207,Z 268.323,A -85,B 0,C 180,E1 -27371.845,E2 -27371.845} C_VEL
LIN {X 0,Y 171.35,Z 268.899,A -85,B 0,C 180,E1 -27373.189,E2 -27373.189} C_VEL
LIN {X 0,Y 172.192,Z 271.816,A -85,B 0,C 180,E1 -27377.213,E2 -27377.213} C_VEL
LIN {X 0,Y 173.411,Z 276.218,A -85,B 0,C 180,E1 -27380.773,E2 -27380.773} C_VEL
LIN {X 0,Y 174.726,Z 281.815,A -85,B 0,C 180,E1 -27383.899,E2 -27383.899} C_VEL
LIN {X 0,Y 174.924,Z 282.854,A -85,B 0,C 180,E1 -27384.385,E2 -27384.385} C_VEL
LIN {X 0,Y 172.035,Z 295.553,A -85,B 0,C 180,E1 -27384.896,E2 -27384.896} C_VEL
LIN {X 0,Y 168.184,Z 307.283,A -85,B 0,C 180,E1 -27385.558,E2 -27385.558} C_VEL
LIN {X 0,Y 162.898,Z 319.302,A -85,B 0,C 180,E1 -27386.461,E2 -27386.461} C_VEL
LIN {X 0,Y 156.731,Z 330.52,A -85,B 0,C 180,E1 -27387.672,E2 -27387.672} C_VEL
LIN {X 0,Y 149.867,Z 340.7,A -85,B 0,C 180,E1 -27389.141,E2 -27389.141} C_VEL
LIN {X 0,Y 143.158,Z 349.055,A -85,B 0,C 180,E1 -27390.781,E2 -27390.781} C_VEL
LIN {X 0,Y 134.57,Z 358.141,A -85,B 0,C 180,E1 -27393.319,E2 -27393.319} C_VEL
LIN {X 0,Y 126.244,Z 365.509,A -85,B 0,C 180,E1 -27396.175,E2 -27396.175} C_VEL
LIN {X 0,Y 118.348,Z 371.459,A -85,B 0,C 180,E1 -27399.466,E2 -27399.466} C_VEL
LIN {X 0,Y 110.955,Z 376.206,A -85,B 0,C 180,E1 -27403.245,E2 -27403.245} C_VEL
LIN {X 0,Y 103.16,Z 380.491,A -85,B 0,C 180,E1 -27408.54,E2 -27408.54} C_VEL
LIN {X 0,Y 96.558,Z 383.318,A -85,B 0,C 180,E1 -27414.388,E2 -27414.388} C_VEL
LIN {X 0,Y 90.365,Z 385.132,A -85,B 0,C 180,E1 -27422.183,E2 -27422.183} C_VEL
LIN {X 0,Y 86.212,Z 385.467,A -85,B 0,C 180,E1 -27430.968,E2 -27430.968} C_VEL
LIN {X 0,Y 84.309,Z 384.235,A -85,B 0,C 180,E1 -27440.402,E2 -27440.402} C_VEL
LIN {X 0,Y 84.169,Z 383.046,A -85,B 0,C 180,E1 -27445.209,E2 -27445.209} C_VEL
LIN {X 0,Y 84.338,Z 381.447,A -85,B 0,C 180,E1 -27449.999,E2 -27449.999} C_VEL
LIN {X 0,Y 84.159,Z 378.051,A -85,B 0,C 180,E1 -27457.195,E2 -27457.195} C_VEL
LIN {X 0,Y 84.954,Z 373.526,A -85,B 0,C 180,E1 -27464.369,E2 -27464.369} C_VEL
LIN {X 0,Y 87.298,Z 366.603,A -85,B 0,C 180,E1 -27472.482,E2 -27472.482} C_VEL
LIN {X 0,Y 90.516,Z 359.05,A -85,B 0,C 180,E1 -27479.03,E2 -27479.03} C_VEL
LIN {X 0,Y 94.121,Z 350.871,A -85,B 0,C 180,E1 -27484.394,E2 -27484.394} C_VEL
LIN {X 0,Y 97.745,Z 343.275,A -85,B 0,C 180,E1 -27488.129,E2 -27488.129} C_VEL
LIN {X 0,Y 102.048,Z 332.757,A -85,B 0,C 180,E1 -27492.18,E2 -27492.18} C_VEL
LIN {X 0,Y 105.115,Z 324.523,A -85,B 0,C 180,E1 -27494.589,E2 -27494.589} C_VEL
LIN {X 0,Y 108.966,Z 312.665,A -85,B 0,C 180,E1 -27497.193,E2 -27497.193} C_VEL
LIN {X 0,Y 112.417,Z 299.267,A -85,B 0,C 180,E1 -27499.234,E2 -27499.234} C_VEL
LIN {X 0,Y 114.782,Z 286.143,A -85,B 0,C 180,E1 -27500.561,E2 -27500.561} C_VEL
LIN {X 0,Y 116.471,Z 269.088,A -85,B 0,C 180,E1 -27501.556,E2 -27501.556} C_VEL
LIN {X 0,Y 118.204,Z 246.217,A -85,B 0,C 180,E1 -27502.72,E2 -27502.72} C_VEL
LIN {X 0,Y 117.69,Z 235.832,A -85,B 0,C 180,E1 -27503.864,E2 -27503.864} C_VEL
LIN {X 0,Y 114.146,Z 224.388,A -85,B 0,C 180,E1 -27506.745,E2 -27506.745} C_VEL
LIN {X 0,Y 113.525,Z 222.694,A -85,B 0,C 180,E1 -27507.255,E2 -27507.255} C_VEL
LIN {X 0,Y 112.227,Z 219.69,A -85,B 0,C 180,E1 -27508.306,E2 -27508.306} C_VEL
LIN {X 0,Y 109.516,Z 216.302,A -85,B 0,C 180,E1 -27510.353,E2 -27510.353} C_VEL
LIN {X 0,Y 104.281,Z 212.529,A -85,B 0,C 180,E1 -27514.536,E2 -27514.536} C_VEL
LIN {X 0,Y 100.354,Z 209.566,A -85,B 0,C 180,E1 -27518.284,E2 -27518.284} C_VEL
LIN {X 0,Y 98.749,Z 207.567,A -85,B 0,C 180,E1 -27520.149,E2 -27520.149} C_VEL
LIN {X 0,Y 97.036,Z 204.839,A -85,B 0,C 180,E1 -27522.446,E2 -27522.446} C_VEL
LIN {X 0,Y 94.659,Z 201.468,A -85,B 0,C 180,E1 -27526.053,E2 -27526.053} C_VEL
LIN {X 0,Y 93.936,Z 200.355,A -85,B 0,C 180,E1 -27527.317,E2 -27527.317} C_VEL
LIN {X 0,Y 91.501,Z 197.278,A -85,B 0,C 180,E1 -27532.153,E2 -27532.153} C_VEL
LIN {X 0,Y 90.595,Z 195.358,A -85,B 0,C 180,E1 -27534.586,E2 -27534.586} C_VEL
LIN {X 0,Y 88.588,Z 193.682,A -85,B 0,C 180,E1 -27541.136,E2 -27541.136} C_VEL
LIN {X 0,Y 87.588,Z 193.084,A -85,B 0,C 180,E1 -27549.234,E2 -27549.234} C_VEL
LIN {X 0,Y 87.978,Z 193.999,A -85,B 0,C 180,E1 -27556.832,E2 -27556.832} C_VEL
LIN {X 0,Y 90.437,Z 195.718,A -85,B 0,C 180,E1 -27565.938,E2 -27565.938} C_VEL
LIN {X 0,Y 91.811,Z 198.516,A -85,B 0,C 180,E1 -27569.523,E2 -27569.523} C_VEL
LIN {X 0,Y 94.378,Z 201.215,A -85,B 0,C 180,E1 -27574.242,E2 -27574.242} C_VEL
LIN {X 0,Y 96.758,Z 204.788,A -85,B 0,C 180,E1 -27577.972,E2 -27577.972} C_VEL
LIN {X 0,Y 97.9,Z 206.417,A -85,B 0,C 180,E1 -27579.529,E2 -27579.529} C_VEL
LIN {X 0,Y 100.612,Z 210.403,A -85,B 0,C 180,E1 -27582.837,E2 -27582.837} C_VEL
LIN {X 0,Y 104.391,Z 216.447,A -85,B 0,C 180,E1 -27586.8,E2 -27586.8} C_VEL
LIN {X 0,Y 108.539,Z 224.091,A -85,B 0,C 180,E1 -27590.599,E2 -27590.599} C_VEL
LIN {X 0,Y 113.269,Z 234.48,A -85,B 0,C 180,E1 -27594.486,E2 -27594.486} C_VEL
LIN {X 0,Y 113.886,Z 236.076,A -85,B 0,C 180,E1 -27594.972,E2 -27594.972} C_VEL
LIN {X 0,Y 110.424,Z 275.312,A -85,B 0,C 180,E1 -27596.986,E2 -27596.986} C_VEL
LIN {X 0,Y 108.301,Z 288.62,A -85,B 0,C 180,E1 -27598.252,E2 -27598.252} C_VEL
LIN {X 0,Y 105.54,Z 300.95,A -85,B 0,C 180,E1 -27600.066,E2 -27600.066} C_VEL
LIN {X 0,Y 102.213,Z 312.145,A -85,B 0,C 180,E1 -27602.348,E2 -27602.348} C_VEL
LIN {X 0,Y 97.839,Z 323.934,A -85,B 0,C 180,E1 -27605.605,E2 -27605.605} C_VEL
LIN {X 0,Y 93.39,Z 334.51,A -85,B 0,C 180,E1 -27609.633,E2 -27609.633} C_VEL
LIN {X 0,Y 89.282,Z 343.164,A -85,B 0,C 180,E1 -27614.008,E2 -27614.008} C_VEL
LIN {X 0,Y 84.652,Z 352.505,A -85,B 0,C 180,E1 -27620.443,E2 -27620.443} C_VEL
LIN {X 0,Y 81.063,Z 360.026,A -85,B 0,C 180,E1 -27627.516,E2 -27627.516} C_VEL
LIN {X 0,Y 78.507,Z 366.042,A -85,B 0,C 180,E1 -27635.137,E2 -27635.137} C_VEL
LIN {X 0,Y 76.933,Z 370.788,A -85,B 0,C 180,E1 -27643.203,E2 -27643.203} C_VEL
LIN {X 0,Y 76.594,Z 374.391,A -85,B 0,C 180,E1 -27651.533,E2 -27651.533} C_VEL
LIN {X 0,Y 77.1,Z 376.189,A -85,B 0,C 180,E1 -27657.116,E2 -27657.116} C_VEL
LIN {X 0,Y 78.273,Z 377.551,A -85,B 0,C 180,E1 -27662.598,E2 -27662.598} C_VEL
LIN {X 0,Y 80.04,Z 378.427,A -85,B 0,C 180,E1 -27667.927,E2 -27667.927} C_VEL
LIN {X 0,Y 82.379,Z 378.863,A -85,B 0,C 180,E1 -27673.041,E2 -27673.041} C_VEL
LIN {X 0,Y 86.401,Z 378.754,A -85,B 0,C 180,E1 -27679.404,E2 -27679.404} C_VEL
LIN {X 0,Y 92.691,Z 377.476,A -85,B 0,C 180,E1 -27686.517,E2 -27686.517} C_VEL
LIN {X 0,Y 97.062,Z 376.111,A -85,B 0,C 180,E1 -27690.331,E2 -27690.331} C_VEL
LIN {X 0,Y 104.074,Z 373.232,A -85,B 0,C 180,E1 -27695.259,E2 -27695.259} C_VEL
LIN {X 0,Y 112.321,Z 368.921,A -85,B 0,C 180,E1 -27699.813,E2 -27699.813} C_VEL
LIN {X 0,Y 121.033,Z 363.263,A -85,B 0,C 180,E1 -27703.68,E2 -27703.68} C_VEL
LIN {X 0,Y 129.871,Z 356.308,A -85,B 0,C 180,E1 -27706.927,E2 -27706.927} C_VEL
LIN {X 0,Y 137.695,Z 349.01,A -85,B 0,C 180,E1 -27709.275,E2 -27709.275} C_VEL
LIN {X 0,Y 146.149,Z 339.488,A -85,B 0,C 180,E1 -27711.533,E2 -27711.533} C_VEL
LIN {X 0,Y 153.061,Z 330.031,A -85,B 0,C 180,E1 -27713.193,E2 -27713.193} C_VEL
LIN {X 0,Y 160.07,Z 318.276,A -85,B 0,C 180,E1 -27714.733,E2 -27714.733} C_VEL
LIN {X 0,Y 165.526,Z 306.607,A -85,B 0,C 180,E1 -27715.826,E2 -27715.826} C_VEL
LIN {X 0,Y 169.837,Z 294.497,A -85,B 0,C 180,E1 -27716.672,E2 -27716.672} C_VEL
LIN {X 0,Y 172.65,Z 283.691,A -85,B 0,C 180,E1 -27717.212,E2 -27717.212} C_VEL
LIN {X 0,Y 171.511,Z 279.525,A -85,B 0,C 180,E1 -27720.734,E2 -27720.734} C_VEL
LIN {X 0,Y 170.996,Z 277.998,A -85,B 0,C 180,E1 -27722.651,E2 -27722.651} C_VEL
LIN {X 0,Y 170.383,Z 275.348,A -85,B 0,C 180,E1 -27726.514,E2 -27726.514} C_VEL
LIN {X 0,Y 170.288,Z 275.388,A -85,B 0,C 180,E1 -27732.212,E2 -27732.212} C_VEL
LIN {X 0,Y 171.012,Z 278.813,A -85,B 0,C 180,E1 -27736.873,E2 -27736.873} C_VEL
LIN {X 0,Y 171.758,Z 282.847,A -85,B 0,C 180,E1 -27740.038,E2 -27740.038} C_VEL
LIN {X 0,Y 172.381,Z 286.637,A -85,B 0,C 180,E1 -27742.249,E2 -27742.249} C_VEL
LIN {X 0,Y 169.426,Z 297.952,A -85,B 0,C 180,E1 -27742.724,E2 -27742.724} C_VEL
LIN {X 0,Y 164.966,Z 310.214,A -85,B 0,C 180,E1 -27743.391,E2 -27743.391} C_VEL
LIN {X 0,Y 159.895,Z 320.995,A -85,B 0,C 180,E1 -27744.21,E2 -27744.21} C_VEL
LIN {X 0,Y 153.593,Z 331.814,A -85,B 0,C 180,E1 -27745.349,E2 -27745.349} C_VEL
LIN {X 0,Y 145.794,Z 342.611,A -85,B 0,C 180,E1 -27746.899,E2 -27746.899} C_VEL
LIN {X 0,Y 138.193,Z 351.404,A -85,B 0,C 180,E1 -27748.683,E2 -27748.683} C_VEL
LIN {X 0,Y 129.364,Z 360.024,A -85,B 0,C 180,E1 -27751.167,E2 -27751.167} C_VEL
LIN {X 0,Y 120.809,Z 366.953,A -85,B 0,C 180,E1 -27754.004,E2 -27754.004} C_VEL
LIN {X 0,Y 111.323,Z 373.357,A -85,B 0,C 180,E1 -27757.893,E2 -27757.893} C_VEL
LIN {X 0,Y 103.783,Z 377.612,A -85,B 0,C 180,E1 -27761.848,E2 -27761.848} C_VEL
LIN {X 0,Y 97.279,Z 380.723,A -85,B 0,C 180,E1 -27766.259,E2 -27766.259} C_VEL
LIN {X 0,Y 90.872,Z 383.163,A -85,B 0,C 180,E1 -27771.777,E2 -27771.777} C_VEL
LIN {X 0,Y 84.126,Z 384.879,A -85,B 0,C 180,E1 -27779.917,E2 -27779.917} C_VEL
LIN {X 0,Y 81.478,Z 385.178,A -85,B 0,C 180,E1 -27784.45,E2 -27784.45} C_VEL
LIN {X 0,Y 78.124,Z 384.594,A -85,B 0,C 180,E1 -27794.342,E2 -27794.342} C_VEL
LIN {X 0,Y 77.107,Z 382.502,A -85,B 0,C 180,E1 -27804.769,E2 -27804.769} C_VEL
LIN {X 0,Y 77.249,Z 380.826,A -85,B 0,C 180,E1 -27809.999,E2 -27809.999} C_VEL
LIN {X 0,Y 77.111,Z 377.329,A -85,B 0,C 180,E1 -27817.857,E2 -27817.857} C_VEL
LIN {X 0,Y 78.071,Z 372.676,A -85,B 0,C 180,E1 -27825.667,E2 -27825.667} C_VEL
LIN {X 0,Y 80.75,Z 365.594,A -85,B 0,C 180,E1 -27834.418,E2 -27834.418} C_VEL
LIN {X 0,Y 84.303,Z 357.884,A -85,B 0,C 180,E1 -27841.401,E2 -27841.401} C_VEL
LIN {X 0,Y 88.562,Z 349.113,A -85,B 0,C 180,E1 -27847.198,E2 -27847.198} C_VEL
LIN {X 0,Y 92.174,Z 341.714,A -85,B 0,C 180,E1 -27850.901,E2 -27850.901} C_VEL
LIN {X 0,Y 96.804,Z 330.825,A -85,B 0,C 180,E1 -27855.059,E2 -27855.059} C_VEL
LIN {X 0,Y 101.315,Z 319.152,A -85,B 0,C 180,E1 -27858.218,E2 -27858.218} C_VEL
LIN {X 0,Y 105.153,Z 306.729,A -85,B 0,C 180,E1 -27860.604,E2 -27860.604} C_VEL
LIN {X 0,Y 108.192,Z 293.808,A -85,B 0,C 180,E1 -27862.308,E2 -27862.308} C_VEL
LIN {X 0,Y 110.22,Z 281.182,A -85,B 0,C 180,E1 -27863.385,E2 -27863.385} C_VEL
LIN {X 0,Y 113.135,Z 246.527,A -85,B 0,C 180,E1 -27865.199,E2 -27865.199} C_VEL
LIN {X 0,Y 112.79,Z 238.347,A -85,B 0,C 180,E1 -27866.157,E2 -27866.157} C_VEL
LIN {X 0,Y 109.766,Z 227.976,A -85,B 0,C 180,E1 -27868.953,E2 -27868.953} C_VEL
LIN {X 0,Y 107.768,Z 222.782,A -85,B 0,C 180,E1 -27870.803,E2 -27870.803} C_VEL
LIN {X 0,Y 103.541,Z 215.086,A -85,B 0,C 180,E1 -27874.797,E2 -27874.797} C_VEL
LIN {X 0,Y 99.901,Z 209.073,A -85,B 0,C 180,E1 -27878.781,E2 -27878.781} C_VEL
LIN {X 0,Y 98.749,Z 207.567,A -85,B 0,C 180,E1 -27880.149,E2 -27880.149} C_VEL
LIN {X 0,Y 96.557,Z 205.039,A -85,B 0,C 180,E1 -27882.98,E2 -27882.98} C_VEL
LIN {X 0,Y 94.293,Z 203.636,A -85,B 0,C 180,E1 -27886.154,E2 -27886.154} C_VEL
LIN {X 0,Y 88.385,Z 201.585,A -85,B 0,C 180,E1 -27898.222,E2 -27898.222} C_VEL
LIN {X 0,Y 87.424,Z 200.611,A -85,B 0,C 180,E1 -27902.303,E2 -27902.303} C_VEL
LIN {X 0,Y 86.679,Z 200.235,A -85,B 0,C 180,E1 -27911.375,E2 -27911.375} C_VEL
LIN {X 0,Y 89.002,Z 202.504,A -85,B 0,C 180,E1 -27924.618,E2 -27924.618} C_VEL
LIN {X 0,Y 90.456,Z 205.456,A -85,B 0,C 180,E1 -27928.733,E2 -27928.733} C_VEL
LIN {X 0,Y 92.452,Z 207.626,A -85,B 0,C 180,E1 -27932.681,E2 -27932.681} C_VEL
LIN {X 0,Y 95.615,Z 212.628,A -85,B 0,C 180,E1 -27937.948,E2 -27937.948} C_VEL
LIN {X 0,Y 98.23,Z 216.77,A -85,B 0,C 180,E1 -27941.457,E2 -27941.457} C_VEL
LIN {X 0,Y 101.455,Z 222.256,A -85,B 0,C 180,E1 -27945.169,E2 -27945.169} C_VEL
LIN {X 0,Y 105.143,Z 229.571,A -85,B 0,C 180,E1 -27948.893,E2 -27948.893} C_VEL
LIN {X 0,Y 108.904,Z 238.235,A -85,B 0,C 180,E1 -27952.324,E2 -27952.324} C_VEL
LIN {X 0,Y 105.474,Z 275.659,A -85,B 0,C 180,E1 -27954.285,E2 -27954.285} C_VEL
LIN {X 0,Y 103.31,Z 288.696,A -85,B 0,C 180,E1 -27955.536,E2 -27955.536} C_VEL
LIN {X 0,Y 100.275,Z 301.509,A -85,B 0,C 180,E1 -27957.435,E2 -27957.435} C_VEL
LIN {X 0,Y 96.447,Z 313.444,A -85,B 0,C 180,E1 -27959.937,E2 -27959.937} C_VEL
LIN {X 0,Y 91.86,Z 325.049,A -85,B 0,C 180,E1 -27963.291,E2 -27963.291} C_VEL
LIN {X 0,Y 87.162,Z 335.457,A -85,B 0,C 180,E1 -27967.481,E2 -27967.481} C_VEL
LIN {X 0,Y 82.348,Z 344.83,A -85,B 0,C 180,E1 -27972.621,E2 -27972.621} C_VEL
LIN {X 0,Y 77.527,Z 353.943,A -85,B 0,C 180,E1 -27979.555,E2 -27979.555} C_VEL
LIN {X 0,Y 73.739,Z 361.234,A -85,B 0,C 180,E1 -27987.27,E2 -27987.27} C_VEL
LIN {X 0,Y 71.144,Z 367.054,A -85,B 0,C 180,E1 -27995.67,E2 -27995.67} C_VEL
LIN {X 0,Y 69.685,Z 371.652,A -85,B 0,C 180,E1 -28004.605,E2 -28004.605} C_VEL
LIN {X 0,Y 69.704,Z 375.445,A -85,B 0,C 180,E1 -28014.848,E2 -28014.848} C_VEL
LIN {X 0,Y 70.445,Z 376.843,A -85,B 0,C 180,E1 -28019.924,E2 -28019.924} C_VEL
LIN {X 0,Y 73.5,Z 378.724,A -85,B 0,C 180,E1 -28030.099,E2 -28030.099} C_VEL
LIN {X 0,Y 76.933,Z 379.246,A -85,B 0,C 180,E1 -28036.956,E2 -28036.956} C_VEL
LIN {X 0,Y 80.756,Z 379.102,A -85,B 0,C 180,E1 -28042.47,E2 -28042.47} C_VEL
LIN {X 0,Y 88.674,Z 377.593,A -85,B 0,C 180,E1 -28050.673,E2 -28050.673} C_VEL
LIN {X 0,Y 93.483,Z 376.114,A -85,B 0,C 180,E1 -28054.445,E2 -28054.445} C_VEL
LIN {X 0,Y 102.387,Z 372.487,A -85,B 0,C 180,E1 -28059.928,E2 -28059.928} C_VEL
LIN {X 0,Y 109.908,Z 368.601,A -85,B 0,C 180,E1 -28063.573,E2 -28063.573} C_VEL
LIN {X 0,Y 118.932,Z 362.893,A -85,B 0,C 180,E1 -28067.172,E2 -28067.172} C_VEL
LIN {X 0,Y 128.362,Z 355.635,A -85,B 0,C 180,E1 -28070.243,E2 -28070.243} C_VEL
LIN {X 0,Y 136.486,Z 348.094,A -85,B 0,C 180,E1 -28072.411,E2 -28072.411} C_VEL
LIN {X 0,Y 144.898,Z 338.633,A -85,B 0,C 180,E1 -28074.434,E2 -28074.434} C_VEL
LIN {X 0,Y 152.35,Z 328.464,A -85,B 0,C 180,E1 -28076.014,E2 -28076.014} C_VEL
LIN {X 0,Y 158.719,Z 317.706,A -85,B 0,C 180,E1 -28077.288,E2 -28077.288} C_VEL
LIN {X 0,Y 164.157,Z 306.126,A -85,B 0,C 180,E1 -28078.28,E2 -28078.28} C_VEL
LIN {X 0,Y 168.695,Z 293.39,A -85,B 0,C 180,E1 -28079.09,E2 -28079.09} C_VEL
LIN {X 0,Y 170.077,Z 288.378,A -85,B 0,C 180,E1 -28079.35,E2 -28079.35} C_VEL
LIN {X 0,Y 169.592,Z 285.397,A -85,B 0,C 180,E1 -28082.079,E2 -28082.079} C_VEL
LIN {X 0,Y 169.059,Z 282.303,A -85,B 0,C 180,E1 -28086.715,E2 -28086.715} C_VEL
LIN {X 0,Y 168.989,Z 282.414,A -85,B 0,C 180,E1 -28092.002,E2 -28092.002} C_VEL
LIN {X 0,Y 169.372,Z 285.336,A -85,B 0,C 180,E1 -28096.111,E2 -28096.111} C_VEL
LIN {X 0,Y 169.792,Z 289.252,A -85,B 0,C 180,E1 -28099.224,E2 -28099.224} C_VEL
LIN {X 0,Y 169.871,Z 290.842,A -85,B 0,C 180,E1 -28100.119,E2 -28100.119} C_VEL
LIN {X 0,Y 165.953,Z 303.326,A -85,B 0,C 180,E1 -28100.611,E2 -28100.611} C_VEL
LIN {X 0,Y 161.055,Z 314.987,A -85,B 0,C 180,E1 -28101.288,E2 -28101.288} C_VEL
LIN {X 0,Y 154.735,Z 326.772,A -85,B 0,C 180,E1 -28102.267,E2 -28102.267} C_VEL
LIN {X 0,Y 147.499,Z 337.49,A -85,B 0,C 180,E1 -28103.476,E2 -28103.476} C_VEL
LIN {X 0,Y 139.58,Z 347.162,A -85,B 0,C 180,E1 -28104.997,E2 -28104.997} C_VEL
LIN {X 0,Y 131.906,Z 355.101,A -85,B 0,C 180,E1 -28106.817,E2 -28106.817} C_VEL
LIN {X 0,Y 122.863,Z 362.945,A -85,B 0,C 180,E1 -28109.268,E2 -28109.268} C_VEL
LIN {X 0,Y 115.565,Z 368.287,A -85,B 0,C 180,E1 -28111.635,E2 -28111.635} C_VEL
LIN {X 0,Y 107.111,Z 373.554,A -85,B 0,C 180,E1 -28114.897,E2 -28114.897} C_VEL
LIN {X 0,Y 99.182,Z 377.688,A -85,B 0,C 180,E1 -28118.788,E2 -28118.788} C_VEL
LIN {X 0,Y 91.684,Z 380.918,A -85,B 0,C 180,E1 -28123.623,E2 -28123.623} C_VEL
LIN {X 0,Y 85.401,Z 383.019,A -85,B 0,C 180,E1 -28128.825,E2 -28128.825} C_VEL
LIN {X 0,Y 78.044,Z 384.627,A -85,B 0,C 180,E1 -28137.294,E2 -28137.294} C_VEL
LIN {X 0,Y 75.109,Z 384.838,A -85,B 0,C 180,E1 -28142.104,E2 -28142.104} C_VEL
LIN {X 0,Y 71.301,Z 384.147,A -85,B 0,C 180,E1 -28152.799,E2 -28152.799} C_VEL
LIN {X 0,Y 70.035,Z 381.945,A -85,B 0,C 180,E1 -28164.24,E2 -28164.24} C_VEL
LIN {X 0,Y 70.161,Z 380.178,A -85,B 0,C 180,E1 -28169.999,E2 -28169.999} C_VEL
LIN {X 0,Y 70.074,Z 376.57,A -85,B 0,C 180,E1 -28178.651,E2 -28178.651} C_VEL
LIN {X 0,Y 71.216,Z 371.795,A -85,B 0,C 180,E1 -28187.22,E2 -28187.22} C_VEL
LIN {X 0,Y 73.734,Z 365.715,A -85,B 0,C 180,E1 -28195.398,E2 -28195.398} C_VEL
LIN {X 0,Y 77.527,Z 358.106,A -85,B 0,C 180,E1 -28202.949,E2 -28202.949} C_VEL
LIN {X 0,Y 81.59,Z 350.249,A -85,B 0,C 180,E1 -28208.7,E2 -28208.7} C_VEL
LIN {X 0,Y 85.564,Z 342.902,A -85,B 0,C 180,E1 -28212.658,E2 -28212.658} C_VEL
LIN {X 0,Y 90.264,Z 332.846,A -85,B 0,C 180,E1 -28216.88,E2 -28216.88} C_VEL
LIN {X 0,Y 94.267,Z 323.252,A -85,B 0,C 180,E1 -28219.833,E2 -28219.833} C_VEL
LIN {X 0,Y 98.537,Z 311.155,A -85,B 0,C 180,E1 -28222.51,E2 -28222.51} C_VEL
LIN {X 0,Y 102.06,Z 298.584,A -85,B 0,C 180,E1 -28224.431,E2 -28224.431} C_VEL
LIN {X 0,Y 104.639,Z 285.727,A -85,B 0,C 180,E1 -28225.725,E2 -28225.725} C_VEL
LIN {X 0,Y 106.467,Z 268.731,A -85,B 0,C 180,E1 -28226.756,E2 -28226.756} C_VEL
LIN {X 0,Y 108.287,Z 247.486,A -85,B 0,C 180,E1 -28227.845,E2 -28227.845} C_VEL
LIN {X 0,Y 108.101,Z 240.741,A -85,B 0,C 180,E1 -28228.66,E2 -28228.66} C_VEL
LIN {X 0,Y 105.105,Z 230.141,A -85,B 0,C 180,E1 -28231.83,E2 -28231.83} C_VEL
LIN {X 0,Y 103.495,Z 226.269,A -85,B 0,C 180,E1 -28233.467,E2 -28233.467} C_VEL
LIN {X 0,Y 99.222,Z 218.233,A -85,B 0,C 180,E1 -28238.123,E2 -28238.123} C_VEL
LIN {X 0,Y 96.692,Z 214.164,A -85,B 0,C 180,E1 -28241.315,E2 -28241.315} C_VEL
LIN {X 0,Y 94.57,Z 210.772,A -85,B 0,C 180,E1 -28244.423,E2 -28244.423} C_VEL
LIN {X 0,Y 92.131,Z 206.887,A -85,B 0,C 180,E1 -28248.732,E2 -28248.732} C_VEL
LIN {X 0,Y 89.753,Z 203.475,A -85,B 0,C 180,E1 -28254.048,E2 -28254.048} C_VEL
LIN {X 0,Y 89.295,Z 202.278,A -85,B 0,C 180,E1 -28255.485,E2 -28255.485} C_VEL
LIN {X 0,Y 88.385,Z 201.585,A -85,B 0,C 180,E1 -28258.222,E2 -28258.222} C_VEL
LIN {X 0,Y 87.701,Z 201.29,A -85,B 0,C 180,E1 -28260.731,E2 -28260.731} C_VEL
LIN {X 0,Y 86.839,Z 202.087,A -85,B 0,C 180,E1 -28264.543,E2 -28264.543} C_VEL
LIN {X 0,Y 86.094,Z 207.708,A -85,B 0,C 180,E1 -28276.035,E2 -28276.035} C_VEL
LIN {X 0,Y 86.455,Z 208.491,A -85,B 0,C 180,E1 -28278.673,E2 -28278.673} C_VEL
LIN {X 0,Y 87.652,Z 209.382,A -85,B 0,C 180,E1 -28283.399,E2 -28283.399} C_VEL
LIN {X 0,Y 89.359,Z 212.646,A -85,B 0,C 180,E1 -28288.476,E2 -28288.476} C_VEL
LIN {X 0,Y 90.702,Z 214.309,A -85,B 0,C 180,E1 -28291.338,E2 -28291.338} C_VEL
LIN {X 0,Y 93.447,Z 218.884,A -85,B 0,C 180,E1 -28296.353,E2 -28296.353} C_VEL
LIN {X 0,Y 95.886,Z 223.055,A -85,B 0,C 180,E1 -28299.973,E2 -28299.973} C_VEL
LIN {X 0,Y 99.245,Z 229.352,A -85,B 0,C 180,E1 -28304.198,E2 -28304.198} C_VEL
LIN {X 0,Y 102.385,Z 236.333,A -85,B 0,C 180,E1 -28307.667,E2 -28307.667} C_VEL
LIN {X 0,Y 104.267,Z 241.071,A -85,B 0,C 180,E1 -28309.586,E2 -28309.586} C_VEL
LIN {X 0,Y 100.814,Z 275.696,A -85,B 0,C 180,E1 -28311.309,E2 -28311.309} C_VEL
LIN {X 0,Y 98.432,Z 289.376,A -85,B 0,C 180,E1 -28312.625,E2 -28312.625} C_VEL
LIN {X 0,Y 95.247,Z 301.979,A -85,B 0,C 180,E1 -28314.502,E2 -28314.502} C_VEL
LIN {X 0,Y 90.893,Z 314.708,A -85,B 0,C 180,E1 -28317.232,E2 -28317.232} C_VEL
LIN {X 0,Y 86.059,Z 326.137,A -85,B 0,C 180,E1 -28320.661,E2 -28320.661} C_VEL
LIN {X 0,Y 81.048,Z 336.366,A -85,B 0,C 180,E1 -28324.994,E2 -28324.994} C_VEL
LIN {X 0,Y 75.458,Z 346.477,A -85,B 0,C 180,E1 -28330.976,E2 -28330.976} C_VEL
LIN {X 0,Y 70.308,Z 355.328,A -85,B 0,C 180,E1 -28338.469,E2 -28338.469} C_VEL
LIN {X 0,Y 66.474,Z 362.378,A -85,B 0,C 180,E1 -28346.971,E2 -28346.971} C_VEL
LIN {X 0,Y 63.69,Z 368.262,A -85,B 0,C 180,E1 -28356.731,E2 -28356.731} C_VEL
LIN {X 0,Y 62.445,Z 372.504,A -85,B 0,C 180,E1 -28366.343,E2 -28366.343} C_VEL
LIN {X 0,Y 62.781,Z 375.826,A -85,B 0,C 180,E1 -28376.603,E2 -28376.603} C_VEL
LIN {X 0,Y 63.959,Z 377.457,A -85,B 0,C 180,E1 -28383.328,E2 -28383.328} C_VEL
LIN {X 0,Y 67.232,Z 379.045,A -85,B 0,C 180,E1 -28392.969,E2 -28392.969} C_VEL
LIN {X 0,Y 71.903,Z 379.606,A -85,B 0,C 180,E1 -28401.44,E2 -28401.44} C_VEL
LIN {X 0,Y 75.832,Z 379.402,A -85,B 0,C 180,E1 -28406.525,E2 -28406.525} C_VEL
LIN {X 0,Y 80.282,Z 378.771,A -85,B 0,C 180,E1 -28411.096,E2 -28411.096} C_VEL
LIN {X 0,Y 86.061,Z 377.425,A -85,B 0,C 180,E1 -28415.902,E2 -28415.902} C_VEL
LIN {X 0,Y 96.032,Z 374.039,A -85,B 0,C 180,E1 -28422.064,E2 -28422.064} C_VEL
LIN {X 0,Y 104.916,Z 369.954,A -85,B 0,C 180,E1 -28426.244,E2 -28426.244} C_VEL
LIN {X 0,Y 114.266,Z 364.53,A -85,B 0,C 180,E1 -28429.768,E2 -28429.768} C_VEL
LIN {X 0,Y 123.984,Z 357.574,A -85,B 0,C 180,E1 -28432.744,E2 -28432.744} C_VEL
LIN {X 0,Y 132.147,Z 350.56,A -85,B 0,C 180,E1 -28434.789,E2 -28434.789} C_VEL
LIN {X 0,Y 140.793,Z 341.642,A -85,B 0,C 180,E1 -28436.71,E2 -28436.71} C_VEL
LIN {X 0,Y 148.537,Z 331.9,A -85,B 0,C 180,E1 -28438.253,E2 -28438.253} C_VEL
LIN {X 0,Y 155.603,Z 320.923,A -85,B 0,C 180,E1 -28439.549,E2 -28439.549} C_VEL
LIN {X 0,Y 161.652,Z 309.181,A -85,B 0,C 180,E1 -28440.528,E2 -28440.528} C_VEL
LIN {X 0,Y 166.132,Z 297.82,A -85,B 0,C 180,E1 -28441.265,E2 -28441.265} C_VEL
LIN {X 0,Y 167.638,Z 293.142,A -85,B 0,C 180,E1 -28441.504,E2 -28441.504} C_VEL
LIN {X 0,Y 167.396,Z 291.457,A -85,B 0,C 180,E1 -28443.585,E2 -28443.585} C_VEL
LIN {X 0,Y 167.304,Z 289.118,A -85,B 0,C 180,E1 -28447.24,E2 -28447.24} C_VEL
LIN {X 0,Y 167.283,Z 289.413,A -85,B 0,C 180,E1 -28451.819,E2 -28451.819} C_VEL
LIN {X 0,Y 167.417,Z 291.83,A -85,B 0,C 180,E1 -28455.387,E2 -28455.387} C_VEL
LIN {X 0,Y 167.501,Z 294.263,A -85,B 0,C 180,E1 -28457.478,E2 -28457.478} C_VEL
LIN {X 0,Y 167.128,Z 296.06,A -85,B 0,C 180,E1 -28457.917,E2 -28457.917} C_VEL
LIN {X 0,Y 162.962,Z 307.55,A -85,B 0,C 180,E1 -28458.415,E2 -28458.415} C_VEL
LIN {X 0,Y 157.114,Z 319.79,A -85,B 0,C 180,E1 -28459.116,E2 -28459.116} C_VEL
LIN {X 0,Y 150.564,Z 330.691,A -85,B 0,C 180,E1 -28460.049,E2 -28460.049} C_VEL
LIN {X 0,Y 143.204,Z 340.596,A -85,B 0,C 180,E1 -28461.177,E2 -28461.177} C_VEL
LIN {X 0,Y 135.176,Z 349.608,A -85,B 0,C 180,E1 -28462.652,E2 -28462.652} C_VEL
LIN {X 0,Y 125.742,Z 358.435,A -85,B 0,C 180,E1 -28464.734,E2 -28464.734} C_VEL
LIN {X 0,Y 116.532,Z 365.572,A -85,B 0,C 180,E1 -28467.18,E2 -28467.18} C_VEL
LIN {X 0,Y 106.104,Z 372.127,A -85,B 0,C 180,E1 -28470.561,E2 -28470.561} C_VEL
LIN {X 0,Y 97.602,Z 376.508,A -85,B 0,C 180,E1 -28474.096,E2 -28474.096} C_VEL
LIN {X 0,Y 89.687,Z 379.862,A -85,B 0,C 180,E1 -28478.406,E2 -28478.406} C_VEL
LIN {X 0,Y 80.174,Z 382.876,A -85,B 0,C 180,E1 -28485.469,E2 -28485.469} C_VEL
LIN {X 0,Y 75.903,Z 383.811,A -85,B 0,C 180,E1 -28489.597,E2 -28489.597} C_VEL
LIN {X 0,Y 68.892,Z 384.486,A -85,B 0,C 180,E1 -28499.33,E2 -28499.33} C_VEL
LIN {X 0,Y 64.535,Z 383.695,A -85,B 0,C 180,E1 -28510.93,E2 -28510.93} C_VEL
LIN {X 0,Y 63.383,Z 382.736,A -85,B 0,C 180,E1 -28517.186,E2 -28517.186} C_VEL
LIN {X 0,Y 62.994,Z 381.35,A -85,B 0,C 180,E1 -28523.593,E2 -28523.593} C_VEL
LIN {X 0,Y 63.06,Z 379.529,A -85,B 0,C 180,E1 -28529.999,E2 -28529.999} C_VEL
LIN {X 0,Y 63.048,Z 375.811,A -85,B 0,C 180,E1 -28539.624,E2 -28539.624} C_VEL
LIN {X 0,Y 64.436,Z 370.916,A -85,B 0,C 180,E1 -28549.098,E2 -28549.098} C_VEL
LIN {X 0,Y 67.363,Z 364.707,A -85,B 0,C 180,E1 -28558,E2 -28558} C_VEL
LIN {X 0,Y 70.843,Z 358.33,A -85,B 0,C 180,E1 -28564.779,E2 -28564.779} C_VEL
LIN {X 0,Y 75.967,Z 349.235,A -85,B 0,C 180,E1 -28571.823,E2 -28571.823} C_VEL
LIN {X 0,Y 80.399,Z 341.355,A -85,B 0,C 180,E1 -28576.15,E2 -28576.15} C_VEL
LIN {X 0,Y 85.486,Z 330.935,A -85,B 0,C 180,E1 -28580.419,E2 -28580.419} C_VEL
LIN {X 0,Y 89.851,Z 321.021,A -85,B 0,C 180,E1 -28583.295,E2 -28583.295} C_VEL
LIN {X 0,Y 94.36,Z 308.406,A -85,B 0,C 180,E1 -28585.954,E2 -28585.954} C_VEL
LIN {X 0,Y 97.69,Z 296.242,A -85,B 0,C 180,E1 -28587.705,E2 -28587.705} C_VEL
LIN {X 0,Y 100.205,Z 283.532,A -85,B 0,C 180,E1 -28588.852,E2 -28588.852} C_VEL
LIN {X 0,Y 102.396,Z 262.643,A -85,B 0,C 180,E1 -28590.017,E2 -28590.017} C_VEL
LIN {X 0,Y 103.689,Z 247.565,A -85,B 0,C 180,E1 -28590.835,E2 -28590.835} C_VEL
LIN {X 0,Y 103.551,Z 242.791,A -85,B 0,C 180,E1 -28591.484,E2 -28591.484} C_VEL
LIN {X 0,Y 100.962,Z 233.282,A -85,B 0,C 180,E1 -28594.59,E2 -28594.59} C_VEL
LIN {X 0,Y 97.708,Z 226.351,A -85,B 0,C 180,E1 -28598.409,E2 -28598.409} C_VEL
LIN {X 0,Y 94.561,Z 220.542,A -85,B 0,C 180,E1 -28602.704,E2 -28602.704} C_VEL
LIN {X 0,Y 92.39,Z 216.915,A -85,B 0,C 180,E1 -28606.216,E2 -28606.216} C_VEL
LIN {X 0,Y 90.216,Z 213.207,A -85,B 0,C 180,E1 -28610.541,E2 -28610.541} C_VEL
LIN {X 0,Y 87.957,Z 209.245,A -85,B 0,C 180,E1 -28616.563,E2 -28616.563} C_VEL
LIN {X 0,Y 86.48,Z 207.643,A -85,B 0,C 180,E1 -28622.473,E2 -28622.473} C_VEL
LIN {X 0,Y 85.767,Z 207.219,A -85,B 0,C 180,E1 -28630.487,E2 -28630.487} C_VEL
LIN {X 0,Y 86.455,Z 208.491,A -85,B 0,C 180,E1 -28638.673,E2 -28638.673} C_VEL
LIN {X 0,Y 86.945,Z 209.45,A -85,B 0,C 180,E1 -28641.16,E2 -28641.16} C_VEL
LIN {X 0,Y 87.721,Z 212.152,A -85,B 0,C 180,E1 -28644.573,E2 -28644.573} C_VEL
LIN {X 0,Y 88.545,Z 215.744,A -85,B 0,C 180,E1 -28647.63,E2 -28647.63} C_VEL
LIN {X 0,Y 90.745,Z 223.719,A -85,B 0,C 180,E1 -28653.478,E2 -28653.478} C_VEL
LIN {X 0,Y 91.816,Z 225.998,A -85,B 0,C 180,E1 -28655.506,E2 -28655.506} C_VEL
LIN {X 0,Y 94.65,Z 231.372,A -85,B 0,C 180,E1 -28659.948,E2 -28659.948} C_VEL
LIN {X 0,Y 97.85,Z 238.487,A -85,B 0,C 180,E1 -28664.195,E2 -28664.195} C_VEL
LIN {X 0,Y 99.768,Z 243.471,A -85,B 0,C 180,E1 -28666.497,E2 -28666.497} C_VEL
LIN {X 0,Y 96.249,Z 276.86,A -85,B 0,C 180,E1 -28668.166,E2 -28668.166} C_VEL
LIN {X 0,Y 93.761,Z 290.189,A -85,B 0,C 180,E1 -28669.456,E2 -28669.456} C_VEL
LIN {X 0,Y 90.728,Z 301.552,A -85,B 0,C 180,E1 -28671.12,E2 -28671.12} C_VEL
LIN {X 0,Y 86.874,Z 312.647,A -85,B 0,C 180,E1 -28673.37,E2 -28673.37} C_VEL
LIN {X 0,Y 81.693,Z 324.516,A -85,B 0,C 180,E1 -28676.741,E2 -28676.741} C_VEL
LIN {X 0,Y 76.258,Z 335.164,A -85,B 0,C 180,E1 -28681.064,E2 -28681.064} C_VEL
LIN {X 0,Y 70.656,Z 344.733,A -85,B 0,C 180,E1 -28686.556,E2 -28686.556} C_VEL
LIN {X 0,Y 65.103,Z 353.683,A -85,B 0,C 180,E1 -28694.023,E2 -28694.023} C_VEL
LIN {X 0,Y 61.024,Z 360.249,A -85,B 0,C 180,E1 -28701.724,E2 -28701.724} C_VEL
LIN {X 0,Y 58.038,Z 365.482,A -85,B 0,C 180,E1 -28710.001,E2 -28710.001} C_VEL
LIN {X 0,Y 55.825,Z 370.575,A -85,B 0,C 180,E1 -28720.886,E2 -28720.886} C_VEL
LIN {X 0,Y 55.358,Z 374.498,A -85,B 0,C 180,E1 -28732.389,E2 -28732.389} C_VEL
LIN {X 0,Y 56.094,Z 376.525,A -85,B 0,C 180,E1 -28740.078,E2 -28740.078} C_VEL
LIN {X 0,Y 57.735,Z 378.035,A -85,B 0,C 180,E1 -28747.493,E2 -28747.493} C_VEL
LIN {X 0,Y 61.133,Z 379.364,A -85,B 0,C 180,E1 -28756.389,E2 -28756.389} C_VEL
LIN {X 0,Y 67.375,Z 379.922,A -85,B 0,C 180,E1 -28766.565,E2 -28766.565} C_VEL
LIN {X 0,Y 71.877,Z 379.652,A -85,B 0,C 180,E1 -28771.644,E2 -28771.644} C_VEL
LIN {X 0,Y 76.841,Z 378.949,A -85,B 0,C 180,E1 -28776.153,E2 -28776.153} C_VEL
LIN {X 0,Y 82.218,Z 377.736,A -85,B 0,C 180,E1 -28780.101,E2 -28780.101} C_VEL
LIN {X 0,Y 90.92,Z 375.049,A -85,B 0,C 180,E1 -28785.072,E2 -28785.072} C_VEL
LIN {X 0,Y 100.176,Z 371.203,A -85,B 0,C 180,E1 -28789.175,E2 -28789.175} C_VEL
LIN {X 0,Y 110.151,Z 365.912,A -85,B 0,C 180,E1 -28792.669,E2 -28792.669} C_VEL
LIN {X 0,Y 119.859,Z 359.522,A -85,B 0,C 180,E1 -28795.426,E2 -28795.426} C_VEL
LIN {X 0,Y 128.396,Z 352.715,A -85,B 0,C 180,E1 -28797.387,E2 -28797.387} C_VEL
LIN {X 0,Y 137.062,Z 344.368,A -85,B 0,C 180,E1 -28799.15,E2 -28799.15} C_VEL
LIN {X 0,Y 145.693,Z 334.243,A -85,B 0,C 180,E1 -28800.7,E2 -28800.7} C_VEL
LIN {X 0,Y 152.944,Z 323.769,A -85,B 0,C 180,E1 -28801.899,E2 -28801.899} C_VEL
LIN {X 0,Y 159.543,Z 311.7,A -85,B 0,C 180,E1 -28802.879,E2 -28802.879} C_VEL
LIN {X 0,Y 164.689,Z 299.462,A -85,B 0,C 180,E1 -28803.634,E2 -28803.634} C_VEL
LIN {X 0,Y 165.106,Z 298.048,A -85,B 0,C 180,E1 -28804.02,E2 -28804.02} C_VEL
LIN {X 0,Y 165.211,Z 295.903,A -85,B 0,C 180,E1 -28807.333,E2 -28807.333} C_VEL
LIN {X 0,Y 165.125,Z 295.883,A -85,B 0,C 180,E1 -28809.803,E2 -28809.803} C_VEL
LIN {X 0,Y 165.143,Z 296.634,A -85,B 0,C 180,E1 -28812.286,E2 -28812.286} C_VEL
LIN {X 0,Y 165.1,Z 298.938,A -85,B 0,C 180,E1 -28815.28,E2 -28815.28} C_VEL
LIN {X 0,Y 164.779,Z 300.182,A -85,B 0,C 180,E1 -28815.609,E2 -28815.609} C_VEL
LIN {X 0,Y 160.017,Z 311.794,A -85,B 0,C 180,E1 -28816.128,E2 -28816.128} C_VEL
LIN {X 0,Y 154.139,Z 322.918,A -85,B 0,C 180,E1 -28816.762,E2 -28816.762} C_VEL
LIN {X 0,Y 146.639,Z 334.304,A -85,B 0,C 180,E1 -28817.719,E2 -28817.719} C_VEL
LIN {X 0,Y 139.178,Z 343.528,A -85,B 0,C 180,E1 -28818.77,E2 -28818.77} C_VEL
LIN {X 0,Y 130.982,Z 351.974,A -85,B 0,C 180,E1 -28820.117,E2 -28820.117} C_VEL
LIN {X 0,Y 121.362,Z 360.225,A -85,B 0,C 180,E1 -28822.095,E2 -28822.095} C_VEL
LIN {X 0,Y 111.887,Z 366.925,A -85,B 0,C 180,E1 -28824.383,E2 -28824.383} C_VEL
LIN {X 0,Y 102.68,Z 372.324,A -85,B 0,C 180,E1 -28827.151,E2 -28827.151} C_VEL
LIN {X 0,Y 93.809,Z 376.585,A -85,B 0,C 180,E1 -28830.506,E2 -28830.506} C_VEL
LIN {X 0,Y 85.442,Z 379.826,A -85,B 0,C 180,E1 -28834.658,E2 -28834.658} C_VEL
LIN {X 0,Y 75.261,Z 382.732,A -85,B 0,C 180,E1 -28841.662,E2 -28841.662} C_VEL
LIN {X 0,Y 66.512,Z 384.041,A -85,B 0,C 180,E1 -28850.653,E2 -28850.653} C_VEL
LIN {X 0,Y 60.005,Z 383.87,A -85,B 0,C 180,E1 -28862.062,E2 -28862.062} C_VEL
LIN {X 0,Y 57.846,Z 383.234,A -85,B 0,C 180,E1 -28868.623,E2 -28868.623} C_VEL
LIN {X 0,Y 55.949,Z 380.736,A -85,B 0,C 180,E1 -28882.782,E2 -28882.782} C_VEL
LIN {X 0,Y 55.971,Z 378.862,A -85,B 0,C 180,E1 -28889.999,E2 -28889.999} C_VEL
LIN {X 0,Y 56.062,Z 375.03,A -85,B 0,C 180,E1 -28900.837,E2 -28900.837} C_VEL
LIN {X 0,Y 57.751,Z 370.01,A -85,B 0,C 180,E1 -28911.412,E2 -28911.412} C_VEL
LIN {X 0,Y 61.153,Z 363.663,A -85,B 0,C 180,E1 -28921.141,E2 -28921.141} C_VEL
LIN {X 0,Y 65.946,Z 355.642,A -85,B 0,C 180,E1 -28929.748,E2 -28929.748} C_VEL
LIN {X 0,Y 71.334,Z 347.018,A -85,B 0,C 180,E1 -28936.103,E2 -28936.103} C_VEL
LIN {X 0,Y 76.804,Z 337.494,A -85,B 0,C 180,E1 -28941.058,E2 -28941.058} C_VEL
LIN {X 0,Y 81.734,Z 327.629,A -85,B 0,C 180,E1 -28944.771,E2 -28944.771} C_VEL
LIN {X 0,Y 86.444,Z 317.008,A -85,B 0,C 180,E1 -28947.51,E2 -28947.51} C_VEL
LIN {X 0,Y 90.933,Z 304.187,A -85,B 0,C 180,E1 -28949.841,E2 -28949.841} C_VEL
LIN {X 0,Y 94.28,Z 291.313,A -85,B 0,C 180,E1 -28951.426,E2 -28951.426} C_VEL
LIN {X 0,Y 96.467,Z 278.397,A -85,B 0,C 180,E1 -28952.403,E2 -28952.403} C_VEL
LIN {X 0,Y 99.355,Z 249.019,A -85,B 0,C 180,E1 -28953.895,E2 -28953.895} C_VEL
LIN {X 0,Y 99.31,Z 245.298,A -85,B 0,C 180,E1 -28954.405,E2 -28954.405} C_VEL
LIN {X 0,Y 97.256,Z 237.221,A -85,B 0,C 180,E1 -28957.284,E2 -28957.284} C_VEL
LIN {X 0,Y 93.759,Z 229.491,A -85,B 0,C 180,E1 -28962.129,E2 -28962.129} C_VEL
LIN {X 0,Y 90.729,Z 223.591,A -85,B 0,C 180,E1 -28967.309,E2 -28967.309} C_VEL
LIN {X 0,Y 88.242,Z 219.284,A -85,B 0,C 180,E1 -28972.759,E2 -28972.759} C_VEL
LIN {X 0,Y 86.4,Z 215.655,A -85,B 0,C 180,E1 -28978.688,E2 -28978.688} C_VEL
LIN {X 0,Y 85.386,Z 214.582,A -85,B 0,C 180,E1 -28983.538,E2 -28983.538} C_VEL
LIN {X 0,Y 84.867,Z 214.306,A -85,B 0,C 180,E1 -28990.927,E2 -28990.927} C_VEL
LIN {X 0,Y 86.392,Z 216.341,A -85,B 0,C 180,E1 -29002.336,E2 -29002.336} C_VEL
LIN {X 0,Y 88.507,Z 220.103,A -85,B 0,C 180,E1 -29008.776,E2 -29008.776} C_VEL
LIN {X 0,Y 91.244,Z 224.906,A -85,B 0,C 180,E1 -29014.476,E2 -29014.476} C_VEL
LIN {X 0,Y 91.816,Z 225.998,A -85,B 0,C 180,E1 -29015.506,E2 -29015.506} C_VEL
LIN {X 0,Y 92.737,Z 228.608,A -85,B 0,C 180,E1 -29017.215,E2 -29017.215} C_VEL
LIN {X 0,Y 93.397,Z 233.188,A -85,B 0,C 180,E1 -29018.82,E2 -29018.82} C_VEL
LIN {X 0,Y 94.291,Z 241.898,A -85,B 0,C 180,E1 -29021.227,E2 -29021.227} C_VEL
LIN {X 0,Y 94.861,Z 244.092,A -85,B 0,C 180,E1 -29022.15,E2 -29022.15} C_VEL
LIN {X 0,Y 95.508,Z 245.925,A -85,B 0,C 180,E1 -29023.06,E2 -29023.06} C_VEL
LIN {X 0,Y 92.219,Z 276.675,A -85,B 0,C 180,E1 -29024.626,E2 -29024.626} C_VEL
LIN {X 0,Y 89.569,Z 290.28,A -85,B 0,C 180,E1 -29025.88,E2 -29025.88} C_VEL
LIN {X 0,Y 86.066,Z 302.698,A -85,B 0,C 180,E1 -29027.674,E2 -29027.674} C_VEL
LIN {X 0,Y 81.397,Z 314.952,A -85,B 0,C 180,E1 -29030.208,E2 -29030.208} C_VEL
LIN {X 0,Y 75.752,Z 326.85,A -85,B 0,C 180,E1 -29033.741,E2 -29033.741} C_VEL
LIN {X 0,Y 70.003,Z 337.068,A -85,B 0,C 180,E1 -29038.193,E2 -29038.193} C_VEL
LIN {X 0,Y 64.083,Z 346.329,A -85,B 0,C 180,E1 -29043.982,E2 -29043.982} C_VEL
LIN {X 0,Y 58.904,Z 353.954,A -85,B 0,C 180,E1 -29050.847,E2 -29050.847} C_VEL
LIN {X 0,Y 53.772,Z 361.465,A -85,B 0,C 180,E1 -29060.599,E2 -29060.599} C_VEL
LIN {X 0,Y 50.035,Z 367.781,A -85,B 0,C 180,E1 -29072.791,E2 -29072.791} C_VEL
LIN {X 0,Y 48.257,Z 372.853,A -85,B 0,C 180,E1 -29086.936,E2 -29086.936} C_VEL
LIN {X 0,Y 48.969,Z 376.354,A -85,B 0,C 180,E1 -29100.561,E2 -29100.561} C_VEL
LIN {X 0,Y 51.888,Z 378.614,A -85,B 0,C 180,E1 -29112.629,E2 -29112.629} C_VEL
LIN {X 0,Y 55.286,Z 379.68,A -85,B 0,C 180,E1 -29120.537,E2 -29120.537} C_VEL
LIN {X 0,Y 58.911,Z 380.151,A -85,B 0,C 180,E1 -29126.628,E2 -29126.628} C_VEL
LIN {X 0,Y 65.658,Z 380.147,A -85,B 0,C 180,E1 -29134.651,E2 -29134.651} C_VEL
LIN {X 0,Y 74.06,Z 379.072,A -85,B 0,C 180,E1 -29141.618,E2 -29141.618} C_VEL
LIN {X 0,Y 79.928,Z 377.787,A -85,B 0,C 180,E1 -29145.292,E2 -29145.292} C_VEL
LIN {X 0,Y 89.251,Z 374.968,A -85,B 0,C 180,E1 -29149.839,E2 -29149.839} C_VEL
LIN {X 0,Y 99.024,Z 370.987,A -85,B 0,C 180,E1 -29153.532,E2 -29153.532} C_VEL
LIN {X 0,Y 109.646,Z 365.413,A -85,B 0,C 180,E1 -29156.703,E2 -29156.703} C_VEL
LIN {X 0,Y 119.493,Z 358.917,A -85,B 0,C 180,E1 -29159.071,E2 -29159.071} C_VEL
LIN {X 0,Y 130.043,Z 350.346,A -85,B 0,C 180,E1 -29161.089,E2 -29161.089} C_VEL
LIN {X 0,Y 138.369,Z 342.058,A -85,B 0,C 180,E1 -29162.518,E2 -29162.518} C_VEL
LIN {X 0,Y 146.136,Z 332.687,A -85,B 0,C 180,E1 -29163.697,E2 -29163.697} C_VEL
LIN {X 0,Y 153.383,Z 321.918,A -85,B 0,C 180,E1 -29164.732,E2 -29164.732} C_VEL
LIN {X 0,Y 159.27,Z 311.029,A -85,B 0,C 180,E1 -29165.468,E2 -29165.468} C_VEL
LIN {X 0,Y 162.509,Z 303.714,A -85,B 0,C 180,E1 -29165.909,E2 -29165.909} C_VEL
LIN {X 0,Y 162.72,Z 302.664,A -85,B 0,C 180,E1 -29167.445,E2 -29167.445} C_VEL
LIN {X 0,Y 162.691,Z 302.601,A -85,B 0,C 180,E1 -29169.951,E2 -29169.951} C_VEL
LIN {X 0,Y 162.611,Z 303.604,A -85,B 0,C 180,E1 -29172.48,E2 -29172.48} C_VEL
LIN {X 0,Y 162.09,Z 305.36,A -85,B 0,C 180,E1 -29173.334,E2 -29173.334} C_VEL
LIN {X 0,Y 156.405,Z 317.342,A -85,B 0,C 180,E1 -29173.84,E2 -29173.84} C_VEL
LIN {X 0,Y 149.722,Z 328.444,A -85,B 0,C 180,E1 -29174.5,E2 -29174.5} C_VEL
LIN {X 0,Y 142.107,Z 338.693,A -85,B 0,C 180,E1 -29175.335,E2 -29175.335} C_VEL
LIN {X 0,Y 133.71,Z 347.938,A -85,B 0,C 180,E1 -29176.412,E2 -29176.412} C_VEL
LIN {X 0,Y 123.808,Z 356.91,A -85,B 0,C 180,E1 -29178.043,E2 -29178.043} C_VEL
LIN {X 0,Y 114.012,Z 364.19,A -85,B 0,C 180,E1 -29179.938,E2 -29179.938} C_VEL
LIN {X 0,Y 102.792,Z 370.923,A -85,B 0,C 180,E1 -29182.628,E2 -29182.628} C_VEL
LIN {X 0,Y 93.439,Z 375.417,A -85,B 0,C 180,E1 -29185.499,E2 -29185.499} C_VEL
LIN {X 0,Y 87.414,Z 377.81,A -85,B 0,C 180,E1 -29187.822,E2 -29187.822} C_VEL
LIN {X 0,Y 76.043,Z 381.382,A -85,B 0,C 180,E1 -29193.715,E2 -29193.715} C_VEL
LIN {X 0,Y 65.712,Z 383.33,A -85,B 0,C 180,E1 -29201.524,E2 -29201.524} C_VEL
LIN {X 0,Y 57.114,Z 383.783,A -85,B 0,C 180,E1 -29212.027,E2 -29212.027} C_VEL
LIN {X 0,Y 53.801,Z 383.462,A -85,B 0,C 180,E1 -29218.497,E2 -29218.497} C_VEL
LIN {X 0,Y 49.645,Z 381.623,A -85,B 0,C 180,E1 -29233.551,E2 -29233.551} C_VEL
LIN {X 0,Y 48.937,Z 380.124,A -85,B 0,C 180,E1 -29241.741,E2 -29241.741} C_VEL
LIN {X 0,Y 48.873,Z 378.193,A -85,B 0,C 180,E1 -29249.998,E2 -29249.998} C_VEL
LIN {X 0,Y 49.071,Z 374.24,A -85,B 0,C 180,E1 -29262.404,E2 -29262.404} C_VEL
LIN {X 0,Y 51.699,Z 368.073,A -85,B 0,C 180,E1 -29276.217,E2 -29276.217} C_VEL
LIN {X 0,Y 55.997,Z 361.3,A -85,B 0,C 180,E1 -29286.594,E2 -29286.594} C_VEL
LIN {X 0,Y 61.655,Z 352.824,A -85,B 0,C 180,E1 -29295.431,E2 -29295.431} C_VEL
LIN {X 0,Y 67.813,Z 343.689,A -85,B 0,C 180,E1 -29301.549,E2 -29301.549} C_VEL
LIN {X 0,Y 73.831,Z 333.339,A -85,B 0,C 180,E1 -29306.398,E2 -29306.398} C_VEL
LIN {X 0,Y 79.244,Z 322.605,A -85,B 0,C 180,E1 -29309.847,E2 -29309.847} C_VEL
LIN {X 0,Y 84.236,Z 310.623,A -85,B 0,C 180,E1 -29312.431,E2 -29312.431} C_VEL
LIN {X 0,Y 88.163,Z 298.656,A -85,B 0,C 180,E1 -29314.16,E2 -29314.16} C_VEL
LIN {X 0,Y 91.284,Z 285.376,A -85,B 0,C 180,E1 -29315.434,E2 -29315.434} C_VEL
LIN {X 0,Y 93.249,Z 270.309,A -85,B 0,C 180,E1 -29316.326,E2 -29316.326} C_VEL
LIN {X 0,Y 95.327,Z 249.753,A -85,B 0,C 180,E1 -29317.316,E2 -29317.316} C_VEL
LIN {X 0,Y 95.221,Z 247.375,A -85,B 0,C 180,E1 -29317.763,E2 -29317.763} C_VEL
LIN {X 0,Y 93.877,Z 241.568,A -85,B 0,C 180,E1 -29320.017,E2 -29320.017} C_VEL
LIN {X 0,Y 90.999,Z 234.669,A -85,B 0,C 180,E1 -29324.684,E2 -29324.684} C_VEL
LIN {X 0,Y 88.645,Z 229.68,A -85,B 0,C 180,E1 -29329.362,E2 -29329.362} C_VEL
LIN {X 0,Y 86.742,Z 225.938,A -85,B 0,C 180,E1 -29334.093,E2 -29334.093} C_VEL
LIN {X 0,Y 85.14,Z 222.46,A -85,B 0,C 180,E1 -29339.999,E2 -29339.999} C_VEL
LIN {X 0,Y 84.303,Z 221.506,A -85,B 0,C 180,E1 -29344.781,E2 -29344.781} C_VEL
LIN {X 0,Y 83.965,Z 221.376,A -85,B 0,C 180,E1 -29351.046,E2 -29351.046} C_VEL
LIN {X 0,Y 85.157,Z 223.208,A -85,B 0,C 180,E1 -29361.176,E2 -29361.176} C_VEL
LIN {X 0,Y 87.361,Z 227.544,A -85,B 0,C 180,E1 -29368.483,E2 -29368.483} C_VEL
LIN {X 0,Y 89.538,Z 231.757,A -85,B 0,C 180,E1 -29373.328,E2 -29373.328} C_VEL
LIN {X 0,Y 92.267,Z 237.517,A -85,B 0,C 180,E1 -29378.213,E2 -29378.213} C_VEL
LIN {X 0,Y 94.809,Z 243.94,A -85,B 0,C 180,E1 -29382.074,E2 -29382.074} C_VEL
LIN {X 0,Y 94.861,Z 244.092,A -85,B 0,C 180,E1 -29382.15,E2 -29382.15} C_VEL
LIN {X 0,Y 95.118,Z 246.269,A -85,B 0,C 180,E1 -29382.731,E2 -29382.731} C_VEL
LIN {X 0,Y 94.697,Z 249.371,A -85,B 0,C 180,E1 -29382.774,E2 -29382.774} C_VEL
LIN {X 0,Y 93.357,Z 253.678,A -85,B 0,C 180,E1 -29382.073,E2 -29382.073} C_VEL
LIN {X 0,Y 90.893,Z 260.308,A -85,B 0,C 180,E1 -29380.477,E2 -29380.477} C_VEL
LIN {X 0,Y 90.084,Z 263.851,A -85,B 0,C 180,E1 -29380.146,E2 -29380.146} C_VEL
LIN {X 0,Y 89.992,Z 264.579,A -85,B 0,C 180,E1 -29380.163,E2 -29380.163} C_VEL
LIN {X 0,Y 87.866,Z 280.581,A -85,B 0,C 180,E1 -29381.031,E2 -29381.031} C_VEL
LIN {X 0,Y 85.011,Z 293.285,A -85,B 0,C 180,E1 -29382.316,E2 -29382.316} C_VEL
LIN {X 0,Y 80.962,Z 305.909,A -85,B 0,C 180,E1 -29384.211,E2 -29384.211} C_VEL
LIN {X 0,Y 75.783,Z 318.183,A -85,B 0,C 180,E1 -29386.849,E2 -29386.849} C_VEL
LIN {X 0,Y 70.085,Z 329.02,A -85,B 0,C 180,E1 -29390.264,E2 -29390.264} C_VEL
LIN {X 0,Y 63.972,Z 338.916,A -85,B 0,C 180,E1 -29394.778,E2 -29394.778} C_VEL
LIN {X 0,Y 57.637,Z 347.934,A -85,B 0,C 180,E1 -29400.809,E2 -29400.809} C_VEL
LIN {X 0,Y 52.02,Z 355.36,A -85,B 0,C 180,E1 -29408.192,E2 -29408.192} C_VEL
LIN {X 0,Y 46.604,Z 362.61,A -85,B 0,C 180,E1 -29419.136,E2 -29419.136} C_VEL
LIN {X 0,Y 43.301,Z 367.577,A -85,B 0,C 180,E1 -29430.002,E2 -29430.002} C_VEL
LIN {X 0,Y 41.231,Z 372.363,A -85,B 0,C 180,E1 -29444.816,E2 -29444.816} C_VEL
LIN {X 0,Y 42.237,Z 376.657,A -85,B 0,C 180,E1 -29463.701,E2 -29463.701} C_VEL
LIN {X 0,Y 46.566,Z 379.192,A -85,B 0,C 180,E1 -29478.995,E2 -29478.995} C_VEL
LIN {X 0,Y 50.434,Z 380.087,A -85,B 0,C 180,E1 -29486.734,E2 -29486.734} C_VEL
LIN {X 0,Y 55.061,Z 380.533,A -85,B 0,C 180,E1 -29493.317,E2 -29493.317} C_VEL
LIN {X 0,Y 61.47,Z 380.5,A -85,B 0,C 180,E1 -29499.942,E2 -29499.942} C_VEL
LIN {X 0,Y 72,Z 379.199,A -85,B 0,C 180,E1 -29507.456,E2 -29507.456} C_VEL
LIN {X 0,Y 78.334,Z 377.852,A -85,B 0,C 180,E1 -29510.721,E2 -29510.721} C_VEL
LIN {X 0,Y 84.879,Z 375.998,A -85,B 0,C 180,E1 -29513.522,E2 -29513.522} C_VEL
LIN {X 0,Y 95.012,Z 372.261,A -85,B 0,C 180,E1 -29516.973,E2 -29516.973} C_VEL
LIN {X 0,Y 106.375,Z 366.743,A -85,B 0,C 180,E1 -29520.001,E2 -29520.001} C_VEL
LIN {X 0,Y 116.037,Z 360.83,A -85,B 0,C 180,E1 -29522.048,E2 -29522.048} C_VEL
LIN {X 0,Y 124.445,Z 354.606,A -85,B 0,C 180,E1 -29523.5,E2 -29523.5} C_VEL
LIN {X 0,Y 134.037,Z 346.052,A -85,B 0,C 180,E1 -29524.967,E2 -29524.967} C_VEL
LIN {X 0,Y 143.156,Z 335.949,A -85,B 0,C 180,E1 -29526.201,E2 -29526.201} C_VEL
LIN {X 0,Y 151.428,Z 324.565,A -85,B 0,C 180,E1 -29527.228,E2 -29527.228} C_VEL
LIN {X 0,Y 157.95,Z 313.126,A -85,B 0,C 180,E1 -29527.935,E2 -29527.935} C_VEL
LIN {X 0,Y 159.886,Z 309.151,A -85,B 0,C 180,E1 -29528.214,E2 -29528.214} C_VEL
LIN {X 0,Y 159.874,Z 309.24,A -85,B 0,C 180,E1 -29530.128,E2 -29530.128} C_VEL
LIN {X 0,Y 159.254,Z 310.751,A -85,B 0,C 180,E1 -29531.007,E2 -29531.007} C_VEL
LIN {X 0,Y 152.977,Z 322.379,A -85,B 0,C 180,E1 -29531.461,E2 -29531.461} C_VEL
LIN {X 0,Y 145.55,Z 333.359,A -85,B 0,C 180,E1 -29532.096,E2 -29532.096} C_VEL
LIN {X 0,Y 136.994,Z 343.56,A -85,B 0,C 180,E1 -29532.905,E2 -29532.905} C_VEL
LIN {X 0,Y 128.512,Z 351.876,A -85,B 0,C 180,E1 -29533.901,E2 -29533.901} C_VEL
LIN {X 0,Y 118.448,Z 360.034,A -85,B 0,C 180,E1 -29535.38,E2 -29535.38} C_VEL
LIN {X 0,Y 108.488,Z 366.646,A -85,B 0,C 180,E1 -29537.15,E2 -29537.15} C_VEL
LIN {X 0,Y 97.039,Z 372.751,A -85,B 0,C 180,E1 -29539.689,E2 -29539.689} C_VEL
LIN {X 0,Y 87.455,Z 376.764,A -85,B 0,C 180,E1 -29542.456,E2 -29542.456} C_VEL
LIN {X 0,Y 78.221,Z 379.773,A -85,B 0,C 180,E1 -29546.039,E2 -29546.039} C_VEL
LIN {X 0,Y 66.642,Z 382.362,A -85,B 0,C 180,E1 -29552.469,E2 -29552.469} C_VEL
LIN {X 0,Y 56.242,Z 383.443,A -85,B 0,C 180,E1 -29561.428,E2 -29561.428} C_VEL
LIN {X 0,Y 51.696,Z 383.43,A -85,B 0,C 180,E1 -29567.174,E2 -29567.174} C_VEL
LIN {X 0,Y 44.897,Z 382.228,A -85,B 0,C 180,E1 -29581.989,E2 -29581.989} C_VEL
LIN {X 0,Y 41.927,Z 379.511,A -85,B 0,C 180,E1 -29600.348,E2 -29600.348} C_VEL
LIN {X 0,Y 41.788,Z 377.491,A -85,B 0,C 180,E1 -29609.998,E2 -29609.998} C_VEL
LIN {X 0,Y 42.136,Z 373.416,A -85,B 0,C 180,E1 -29624.487,E2 -29624.487} C_VEL
LIN {X 0,Y 45.395,Z 367.089,A -85,B 0,C 180,E1 -29640.207,E2 -29640.207} C_VEL
LIN {X 0,Y 50.427,Z 360.169,A -85,B 0,C 180,E1 -29651.451,E2 -29651.451} C_VEL
LIN {X 0,Y 55.686,Z 353.044,A -85,B 0,C 180,E1 -29659.22,E2 -29659.22} C_VEL
LIN {X 0,Y 62.094,Z 344.349,A -85,B 0,C 180,E1 -29665.373,E2 -29665.373} C_VEL
LIN {X 0,Y 68.716,Z 333.86,A -85,B 0,C 180,E1 -29670.38,E2 -29670.38} C_VEL
LIN {X 0,Y 74.424,Z 323.3,A -85,B 0,C 180,E1 -29673.777,E2 -29673.777} C_VEL
LIN {X 0,Y 79.673,Z 311.726,A -85,B 0,C 180,E1 -29676.229,E2 -29676.229} C_VEL
LIN {X 0,Y 84.046,Z 299.181,A -85,B 0,C 180,E1 -29678.002,E2 -29678.002} C_VEL
LIN {X 0,Y 87.322,Z 286.039,A -85,B 0,C 180,E1 -29679.237,E2 -29679.237} C_VEL
LIN {X 0,Y 89.371,Z 272.091,A -85,B 0,C 180,E1 -29680.039,E2 -29680.039} C_VEL
LIN {X 0,Y 91.645,Z 250.43,A -85,B 0,C 180,E1 -29681.059,E2 -29681.059} C_VEL
LIN {X 0,Y 90.714,Z 245.925,A -85,B 0,C 180,E1 -29682.963,E2 -29682.963} C_VEL
LIN {X 0,Y 88.306,Z 239.502,A -85,B 0,C 180,E1 -29687.667,E2 -29687.667} C_VEL
LIN {X 0,Y 86.405,Z 235.226,A -85,B 0,C 180,E1 -29692.133,E2 -29692.133} C_VEL
LIN {X 0,Y 85.152,Z 232.314,A -85,B 0,C 180,E1 -29695.932,E2 -29695.932} C_VEL
LIN {X 0,Y 84.013,Z 229.35,A -85,B 0,C 180,E1 -29700.926,E2 -29700.926} C_VEL
LIN {X 0,Y 83.391,Z 228.545,A -85,B 0,C 180,E1 -29704.834,E2 -29704.834} C_VEL
LIN {X 0,Y 83.062,Z 228.453,A -85,B 0,C 180,E1 -29711.168,E2 -29711.168} C_VEL
LIN {X 0,Y 83.944,Z 230.017,A -85,B 0,C 180,E1 -29719.891,E2 -29719.891} C_VEL
LIN {X 0,Y 85.697,Z 233.925,A -85,B 0,C 180,E1 -29726.721,E2 -29726.721} C_VEL
LIN {X 0,Y 88.059,Z 238.981,A -85,B 0,C 180,E1 -29732.565,E2 -29732.565} C_VEL
LIN {X 0,Y 90.43,Z 244.966,A -85,B 0,C 180,E1 -29737.242,E2 -29737.242} C_VEL
LIN {X 0,Y 91.648,Z 248.502,A -85,B 0,C 180,E1 -29739.368,E2 -29739.368} C_VEL
LIN {X 0,Y 91.139,Z 254.096,A -85,B 0,C 180,E1 -29739.722,E2 -29739.722} C_VEL
LIN {X 0,Y 89.992,Z 264.579,A -85,B 0,C 180,E1 -29740.163,E2 -29740.163} C_VEL
LIN {X 0,Y 89.031,Z 270.408,A -85,B 0,C 180,E1 -29740.04,E2 -29740.04} C_VEL
LIN {X 0,Y 86.283,Z 279.795,A -85,B 0,C 180,E1 -29738.904,E2 -29738.904} C_VEL
LIN {X 0,Y 83.036,Z 289.045,A -85,B 0,C 180,E1 -29737.958,E2 -29737.958} C_VEL
LIN {X 0,Y 81.234,Z 294.652,A -85,B 0,C 180,E1 -29738.19,E2 -29738.19} C_VEL
LIN {X 0,Y 76.986,Z 307.036,A -85,B 0,C 180,E1 -29739.946,E2 -29739.946} C_VEL
LIN {X 0,Y 72.225,Z 317.761,A -85,B 0,C 180,E1 -29742.102,E2 -29742.102} C_VEL
LIN {X 0,Y 66.159,Z 328.777,A -85,B 0,C 180,E1 -29745.272,E2 -29745.272} C_VEL
LIN {X 0,Y 58.902,Z 339.767,A -85,B 0,C 180,E1 -29750.111,E2 -29750.111} C_VEL
LIN {X 0,Y 51.438,Z 349.475,A -85,B 0,C 180,E1 -29756.873,E2 -29756.873} C_VEL
LIN {X 0,Y 44.303,Z 357.952,A -85,B 0,C 180,E1 -29766.637,E2 -29766.637} C_VEL
LIN {X 0,Y 38.588,Z 364.797,A -85,B 0,C 180,E1 -29779.508,E2 -29779.508} C_VEL
LIN {X 0,Y 34.755,Z 370.608,A -85,B 0,C 180,E1 -29797.1,E2 -29797.1} C_VEL
LIN {X 0,Y 34.098,Z 374.515,A -85,B 0,C 180,E1 -29814.347,E2 -29814.347} C_VEL
LIN {X 0,Y 35.684,Z 376.952,A -85,B 0,C 180,E1 -29828.022,E2 -29828.022} C_VEL
LIN {X 0,Y 38.098,Z 378.45,A -85,B 0,C 180,E1 -29837.555,E2 -29837.555} C_VEL
LIN {X 0,Y 44.846,Z 380.305,A -85,B 0,C 180,E1 -29851.958,E2 -29851.958} C_VEL
LIN {X 0,Y 52.059,Z 380.915,A -85,B 0,C 180,E1 -29860.913,E2 -29860.913} C_VEL
LIN {X 0,Y 57.947,Z 380.85,A -85,B 0,C 180,E1 -29865.997,E2 -29865.997} C_VEL
LIN {X 0,Y 64.201,Z 380.304,A -85,B 0,C 180,E1 -29870.144,E2 -29870.144} C_VEL
LIN {X 0,Y 72.731,Z 378.948,A -85,B 0,C 180,E1 -29874.456,E2 -29874.456} C_VEL
LIN {X 0,Y 84.359,Z 375.929,A -85,B 0,C 180,E1 -29878.71,E2 -29878.71} C_VEL
LIN {X 0,Y 94.916,Z 372.051,A -85,B 0,C 180,E1 -29881.599,E2 -29881.599} C_VEL
LIN {X 0,Y 105.669,Z 366.898,A -85,B 0,C 180,E1 -29883.926,E2 -29883.926} C_VEL
LIN {X 0,Y 116.56,Z 360.281,A -85,B 0,C 180,E1 -29885.801,E2 -29885.801} C_VEL
LIN {X 0,Y 127.528,Z 351.864,A -85,B 0,C 180,E1 -29887.263,E2 -29887.263} C_VEL
LIN {X 0,Y 137.368,Z 342.51,A -85,B 0,C 180,E1 -29888.465,E2 -29888.465} C_VEL
LIN {X 0,Y 142.314,Z 336.898,A -85,B 0,C 180,E1 -29889.002,E2 -29889.002} C_VEL
LIN {X 0,Y 142.507,Z 336.704,A -85,B 0,C 180,E1 -29889.479,E2 -29889.479} C_VEL
LIN {X 0,Y 133.875,Z 346.222,A -85,B 0,C 180,E1 -29890.159,E2 -29890.159} C_VEL
LIN {X 0,Y 125.291,Z 354.046,A -85,B 0,C 180,E1 -29890.995,E2 -29890.995} C_VEL
LIN {X 0,Y 115.067,Z 361.727,A -85,B 0,C 180,E1 -29892.245,E2 -29892.245} C_VEL
LIN {X 0,Y 104.923,Z 367.936,A -85,B 0,C 180,E1 -29893.77,E2 -29893.77} C_VEL
LIN {X 0,Y 94.885,Z 372.916,A -85,B 0,C 180,E1 -29895.655,E2 -29895.655} C_VEL
LIN {X 0,Y 84.999,Z 376.809,A -85,B 0,C 180,E1 -29898.034,E2 -29898.034} C_VEL
LIN {X 0,Y 75.373,Z 379.723,A -85,B 0,C 180,E1 -29901.18,E2 -29901.18} C_VEL
LIN {X 0,Y 63.102,Z 382.174,A -85,B 0,C 180,E1 -29906.998,E2 -29906.998} C_VEL
LIN {X 0,Y 51.805,Z 383.142,A -85,B 0,C 180,E1 -29915.511,E2 -29915.511} C_VEL
LIN {X 0,Y 42.302,Z 382.557,A -85,B 0,C 180,E1 -29928.349,E2 -29928.349} C_VEL
LIN {X 0,Y 36.235,Z 380.504,A -85,B 0,C 180,E1 -29947.173,E2 -29947.173} C_VEL
LIN {X 0,Y 34.698,Z 377.874,A -85,B 0,C 180,E1 -29964.185,E2 -29964.185} C_VEL
LIN {X 0,Y 34.704,Z 376.766,A -85,B 0,C 180,E1 -29969.998,E2 -29969.998} C_VEL
LIN {X 0,Y 35.294,Z 372.567,A -85,B 0,C 180,E1 -29987.377,E2 -29987.377} C_VEL
LIN {X 0,Y 39.391,Z 366.108,A -85,B 0,C 180,E1 -30005.438,E2 -30005.438} C_VEL
LIN {X 0,Y 45.309,Z 359.009,A -85,B 0,C 180,E1 -30017.456,E2 -30017.456} C_VEL
LIN {X 0,Y 52.606,Z 350.053,A -85,B 0,C 180,E1 -30026.611,E2 -30026.611} C_VEL
LIN {X 0,Y 59.634,Z 340.907,A -85,B 0,C 180,E1 -30032.148,E2 -30032.148} C_VEL
LIN {X 0,Y 66.2,Z 330.76,A -85,B 0,C 180,E1 -30036.297,E2 -30036.297} C_VEL
LIN {X 0,Y 72.358,Z 319.49,A -85,B 0,C 180,E1 -30039.202,E2 -30039.202} C_VEL
LIN {X 0,Y 77.858,Z 306.815,A -85,B 0,C 180,E1 -30041.403,E2 -30041.403} C_VEL
LIN {X 0,Y 81.826,Z 294.62,A -85,B 0,C 180,E1 -30042.769,E2 -30042.769} C_VEL
LIN {X 0,Y 84.864,Z 281.11,A -85,B 0,C 180,E1 -30043.7,E2 -30043.7} C_VEL
LIN {X 0,Y 88.273,Z 252.538,A -85,B 0,C 180,E1 -30044.973,E2 -30044.973} C_VEL
LIN {X 0,Y 87.684,Z 249.905,A -85,B 0,C 180,E1 -30046.381,E2 -30046.381} C_VEL
LIN {X 0,Y 85.854,Z 244.418,A -85,B 0,C 180,E1 -30050.774,E2 -30050.774} C_VEL
LIN {X 0,Y 83.871,Z 239.151,A -85,B 0,C 180,E1 -30056.993,E2 -30056.993} C_VEL
LIN {X 0,Y 82.785,Z 236.038,A -85,B 0,C 180,E1 -30062.626,E2 -30062.626} C_VEL
LIN {X 0,Y 82.307,Z 235.522,A -85,B 0,C 180,E1 -30066.508,E2 -30066.508} C_VEL
LIN {X 0,Y 82.167,Z 235.623,A -85,B 0,C 180,E1 -30072.015,E2 -30072.015} C_VEL
LIN {X 0,Y 82.797,Z 236.858,A -85,B 0,C 180,E1 -30078.707,E2 -30078.707} C_VEL
LIN {X 0,Y 84.277,Z 240.71,A -85,B 0,C 180,E1 -30085.449,E2 -30085.449} C_VEL
LIN {X 0,Y 85.984,Z 244.969,A -85,B 0,C 180,E1 -30090.388,E2 -30090.388} C_VEL
LIN {X 0,Y 87.891,Z 250.325,A -85,B 0,C 180,E1 -30094.757,E2 -30094.757} C_VEL
LIN {X 0,Y 88.218,Z 251.83,A -85,B 0,C 180,E1 -30095.546,E2 -30095.546} C_VEL
LIN {X 0,Y 84.995,Z 278.272,A -85,B 0,C 180,E1 -30096.717,E2 -30096.717} C_VEL
LIN {X 0,Y 82.107,Z 291.558,A -85,B 0,C 180,E1 -30097.83,E2 -30097.83} C_VEL
LIN {X 0,Y 81.234,Z 294.652,A -85,B 0,C 180,E1 -30098.19,E2 -30098.19} C_VEL
LIN {X 0,Y 79.197,Z 300.255,A -85,B 0,C 180,E1 -30098.495,E2 -30098.495} C_VEL
LIN {X 0,Y 74.583,Z 309.061,A -85,B 0,C 180,E1 -30097.928,E2 -30097.928} C_VEL
LIN {X 0,Y 69.377,Z 317.465,A -85,B 0,C 180,E1 -30097.432,E2 -30097.432} C_VEL
LIN {X 0,Y 66.394,Z 322.44,A -85,B 0,C 180,E1 -30098.033,E2 -30098.033} C_VEL
LIN {X 0,Y 59.689,Z 333.218,A -85,B 0,C 180,E1 -30101.358,E2 -30101.358} C_VEL
LIN {X 0,Y 52.785,Z 342.463,A -85,B 0,C 180,E1 -30105.655,E2 -30105.655} C_VEL
LIN {X 0,Y 45.514,Z 350.931,A -85,B 0,C 180,E1 -30111.857,E2 -30111.857} C_VEL
LIN {X 0,Y 37.709,Z 359.216,A -85,B 0,C 180,E1 -30122.231,E2 -30122.231} C_VEL
LIN {X 0,Y 31.358,Z 365.861,A -85,B 0,C 180,E1 -30137.051,E2 -30137.051} C_VEL
LIN {X 0,Y 27.466,Z 371.207,A -85,B 0,C 180,E1 -30157.601,E2 -30157.601} C_VEL
LIN {X 0,Y 27.399,Z 375.27,A -85,B 0,C 180,E1 -30180.868,E2 -30180.868} C_VEL
LIN {X 0,Y 29.645,Z 377.398,A -85,B 0,C 180,E1 -30195.337,E2 -30195.337} C_VEL
LIN {X 0,Y 33.432,Z 379.063,A -85,B 0,C 180,E1 -30207.236,E2 -30207.236} C_VEL
LIN {X 0,Y 40.484,Z 380.604,A -85,B 0,C 180,E1 -30219.686,E2 -30219.686} C_VEL
LIN {X 0,Y 50.076,Z 381.286,A -85,B 0,C 180,E1 -30229.252,E2 -30229.252} C_VEL
LIN {X 0,Y 56.579,Z 381.106,A -85,B 0,C 180,E1 -30233.589,E2 -30233.589} C_VEL
LIN {X 0,Y 63.338,Z 380.497,A -85,B 0,C 180,E1 -30237.04,E2 -30237.04} C_VEL
LIN {X 0,Y 70.893,Z 379.326,A -85,B 0,C 180,E1 -30240.001,E2 -30240.001} C_VEL
LIN {X 0,Y 80.935,Z 376.957,A -85,B 0,C 180,E1 -30243.009,E2 -30243.009} C_VEL
LIN {X 0,Y 91.787,Z 373.325,A -85,B 0,C 180,E1 -30245.496,E2 -30245.496} C_VEL
LIN {X 0,Y 104.498,Z 367.549,A -85,B 0,C 180,E1 -30247.731,E2 -30247.731} C_VEL
LIN {X 0,Y 109.954,Z 364.53,A -85,B 0,C 180,E1 -30248.516,E2 -30248.516} C_VEL
LIN {X 0,Y 106.9,Z 366.372,A -85,B 0,C 180,E1 -30249.54,E2 -30249.54} C_VEL
LIN {X 0,Y 96.627,Z 371.611,A -85,B 0,C 180,E1 -30250.914,E2 -30250.914} C_VEL
LIN {X 0,Y 86.44,Z 375.722,A -85,B 0,C 180,E1 -30252.662,E2 -30252.662} C_VEL
LIN {X 0,Y 79.722,Z 377.907,A -85,B 0,C 180,E1 -30254.131,E2 -30254.131} C_VEL
LIN {X 0,Y 66.599,Z 381.006,A -85,B 0,C 180,E1 -30258.237,E2 -30258.237} C_VEL
LIN {X 0,Y 53.985,Z 382.595,A -85,B 0,C 180,E1 -30264.311,E2 -30264.311} C_VEL
LIN {X 0,Y 42.391,Z 382.627,A -85,B 0,C 180,E1 -30274.006,E2 -30274.006} C_VEL
LIN {X 0,Y 33.02,Z 381.201,A -85,B 0,C 180,E1 -30290.316,E2 -30290.316} C_VEL
LIN {X 0,Y 29.826,Z 379.92,A -85,B 0,C 180,E1 -30301.88,E2 -30301.88} C_VEL
LIN {X 0,Y 27.691,Z 377.2,A -85,B 0,C 180,E1 -30322.707,E2 -30322.707} C_VEL
LIN {X 0,Y 27.617,Z 376.033,A -85,B 0,C 180,E1 -30329.997,E2 -30329.997} C_VEL
LIN {X 0,Y 28.566,Z 371.71,A -85,B 0,C 180,E1 -30351.653,E2 -30351.653} C_VEL
LIN {X 0,Y 32.851,Z 366.14,A -85,B 0,C 180,E1 -30369.924,E2 -30369.924} C_VEL
LIN {X 0,Y 39.545,Z 359.149,A -85,B 0,C 180,E1 -30383.103,E2 -30383.103} C_VEL
LIN {X 0,Y 46.159,Z 351.945,A -85,B 0,C 180,E1 -30391.099,E2 -30391.099} C_VEL
LIN {X 0,Y 54.65,Z 341.908,A -85,B 0,C 180,E1 -30397.305,E2 -30397.305} C_VEL
LIN {X 0,Y 62.078,Z 331.313,A -85,B 0,C 180,E1 -30401.466,E2 -30401.466} C_VEL
LIN {X 0,Y 68.504,Z 320.276,A -85,B 0,C 180,E1 -30404.109,E2 -30404.109} C_VEL
LIN {X 0,Y 73.825,Z 308.905,A -85,B 0,C 180,E1 -30405.886,E2 -30405.886} C_VEL
LIN {X 0,Y 78.368,Z 296.201,A -85,B 0,C 180,E1 -30407.225,E2 -30407.225} C_VEL
LIN {X 0,Y 81.609,Z 283.139,A -85,B 0,C 180,E1 -30408.072,E2 -30408.072} C_VEL
LIN {X 0,Y 83.907,Z 266.763,A -85,B 0,C 180,E1 -30408.767,E2 -30408.767} C_VEL
LIN {X 0,Y 85.27,Z 255.031,A -85,B 0,C 180,E1 -30409.2,E2 -30409.2} C_VEL
LIN {X 0,Y 83.866,Z 250.192,A -85,B 0,C 180,E1 -30413.274,E2 -30413.274} C_VEL
LIN {X 0,Y 82.466,Z 245.681,A -85,B 0,C 180,E1 -30418.736,E2 -30418.736} C_VEL
LIN {X 0,Y 81.699,Z 242.884,A -85,B 0,C 180,E1 -30423.797,E2 -30423.797} C_VEL
LIN {X 0,Y 81.255,Z 242.468,A -85,B 0,C 180,E1 -30429.96,E2 -30429.96} C_VEL
LIN {X 0,Y 81.712,Z 243.845,A -85,B 0,C 180,E1 -30437.743,E2 -30437.743} C_VEL
LIN {X 0,Y 82.745,Z 247.074,A -85,B 0,C 180,E1 -30443.513,E2 -30443.513} C_VEL
LIN {X 0,Y 84.154,Z 251.28,A -85,B 0,C 180,E1 -30448.447,E2 -30448.447} C_VEL
LIN {X 0,Y 85.135,Z 254.51,A -85,B 0,C 180,E1 -30451.213,E2 -30451.213} C_VEL
LIN {X 0,Y 82.171,Z 278.333,A -85,B 0,C 180,E1 -30452.262,E2 -30452.262} C_VEL
LIN {X 0,Y 79.218,Z 291.481,A -85,B 0,C 180,E1 -30453.222,E2 -30453.222} C_VEL
LIN {X 0,Y 75.5,Z 303.025,A -85,B 0,C 180,E1 -30454.538,E2 -30454.538} C_VEL
LIN {X 0,Y 69.996,Z 315.643,A -85,B 0,C 180,E1 -30456.561,E2 -30456.561} C_VEL
LIN {X 0,Y 66.394,Z 322.44,A -85,B 0,C 180,E1 -30458.033,E2 -30458.033} C_VEL
LIN {X 0,Y 63.24,Z 327.376,A -85,B 0,C 180,E1 -30458.784,E2 -30458.784} C_VEL
LIN {X 0,Y 56.901,Z 335.019,A -85,B 0,C 180,E1 -30458.832,E2 -30458.832} C_VEL
LIN {X 0,Y 49.978,Z 342.142,A -85,B 0,C 180,E1 -30459.177,E2 -30459.177} C_VEL
LIN {X 0,Y 45.94,Z 346.264,A -85,B 0,C 180,E1 -30460.783,E2 -30460.783} C_VEL
LIN {X 0,Y 36.718,Z 355.563,A -85,B 0,C 180,E1 -30468.795,E2 -30468.795} C_VEL
LIN {X 0,Y 28.833,Z 362.742,A -85,B 0,C 180,E1 -30480.826,E2 -30480.826} C_VEL
LIN {X 0,Y 22.453,Z 368.685,A -85,B 0,C 180,E1 -30500.616,E2 -30500.616} C_VEL
LIN {X 0,Y 19.818,Z 373.508,A -85,B 0,C 180,E1 -30530.775,E2 -30530.775} C_VEL
LIN {X 0,Y 23.586,Z 377.494,A -85,B 0,C 180,E1 -30563.425,E2 -30563.425} C_VEL
LIN {X 0,Y 29.986,Z 379.633,A -85,B 0,C 180,E1 -30579.642,E2 -30579.642} C_VEL
LIN {X 0,Y 37.089,Z 380.907,A -85,B 0,C 180,E1 -30589.079,E2 -30589.079} C_VEL
LIN {X 0,Y 49.225,Z 381.608,A -85,B 0,C 180,E1 -30598.088,E2 -30598.088} C_VEL
LIN {X 0,Y 56.242,Z 381.362,A -85,B 0,C 180,E1 -30601.417,E2 -30601.417} C_VEL
LIN {X 0,Y 63.408,Z 380.69,A -85,B 0,C 180,E1 -30604.003,E2 -30604.003} C_VEL
LIN {X 0,Y 70.671,Z 379.519,A -85,B 0,C 180,E1 -30606.016,E2 -30606.016} C_VEL
LIN {X 0,Y 80.358,Z 377.289,A -85,B 0,C 180,E1 -30608.146,E2 -30608.146} C_VEL
LIN {X 0,Y 78.291,Z 377.89,A -85,B 0,C 180,E1 -30609.083,E2 -30609.083} C_VEL
LIN {X 0,Y 64.726,Z 380.875,A -85,B 0,C 180,E1 -30612.244,E2 -30612.244} C_VEL
LIN {X 0,Y 58.039,Z 381.794,A -85,B 0,C 180,E1 -30614.362,E2 -30614.362} C_VEL
LIN {X 0,Y 45.042,Z 382.444,A -85,B 0,C 180,E1 -30620.574,E2 -30620.574} C_VEL
LIN {X 0,Y 33.041,Z 381.63,A -85,B 0,C 180,E1 -30631.695,E2 -30631.695} C_VEL
LIN {X 0,Y 27.906,Z 380.67,A -85,B 0,C 180,E1 -30640.924,E2 -30640.924} C_VEL
LIN {X 0,Y 21.267,Z 377.513,A -85,B 0,C 180,E1 -30670.7,E2 -30670.7} C_VEL
LIN {X 0,Y 20.516,Z 375.281,A -85,B 0,C 180,E1 -30689.996,E2 -30689.996} C_VEL
LIN {X 0,Y 22.082,Z 370.825,A -85,B 0,C 180,E1 -30718.513,E2 -30718.513} C_VEL
LIN {X 0,Y 27.764,Z 365.118,A -85,B 0,C 180,E1 -30739.407,E2 -30739.407} C_VEL
LIN {X 0,Y 35.706,Z 357.9,A -85,B 0,C 180,E1 -30752.338,E2 -30752.338} C_VEL
LIN {X 0,Y 43.16,Z 350.506,A -85,B 0,C 180,E1 -30759.434,E2 -30759.434} C_VEL
LIN {X 0,Y 51.335,Z 341.403,A -85,B 0,C 180,E1 -30764.107,E2 -30764.107} C_VEL
LIN {X 0,Y 58.527,Z 331.741,A -85,B 0,C 180,E1 -30767.327,E2 -30767.327} C_VEL
LIN {X 0,Y 65.214,Z 320.946,A -85,B 0,C 180,E1 -30769.537,E2 -30769.537} C_VEL
LIN {X 0,Y 71.142,Z 308.85,A -85,B 0,C 180,E1 -30771.063,E2 -30771.063} C_VEL
LIN {X 0,Y 75.822,Z 296.217,A -85,B 0,C 180,E1 -30772.145,E2 -30772.145} C_VEL
LIN {X 0,Y 79.146,Z 283.417,A -85,B 0,C 180,E1 -30772.816,E2 -30772.816} C_VEL
LIN {X 0,Y 81.5,Z 267.56,A -85,B 0,C 180,E1 -30773.378,E2 -30773.378} C_VEL
LIN {X 0,Y 82.593,Z 258.211,A -85,B 0,C 180,E1 -30773.741,E2 -30773.741} C_VEL
LIN {X 0,Y 81.616,Z 254.195,A -85,B 0,C 180,E1 -30777.86,E2 -30777.86} C_VEL
LIN {X 0,Y 80.881,Z 251.19,A -85,B 0,C 180,E1 -30782.352,E2 -30782.352} C_VEL
LIN {X 0,Y 80.653,Z 249.684,A -85,B 0,C 180,E1 -30784.998,E2 -30784.998} C_VEL
LIN {X 0,Y 80.349,Z 249.727,A -85,B 0,C 180,E1 -30791.55,E2 -30791.55} C_VEL
LIN {X 0,Y 80.657,Z 250.808,A -85,B 0,C 180,E1 -30796.779,E2 -30796.779} C_VEL
LIN {X 0,Y 81.361,Z 253.596,A -85,B 0,C 180,E1 -30801.762,E2 -30801.762} C_VEL
LIN {X 0,Y 82.394,Z 257.437,A -85,B 0,C 180,E1 -30806.297,E2 -30806.297} C_VEL
LIN {X 0,Y 82.518,Z 257.953,A -85,B 0,C 180,E1 -30806.769,E2 -30806.769} C_VEL
LIN {X 0,Y 79.724,Z 279.033,A -85,B 0,C 180,E1 -30807.548,E2 -30807.548} C_VEL
LIN {X 0,Y 76.545,Z 292.505,A -85,B 0,C 180,E1 -30808.385,E2 -30808.385} C_VEL
LIN {X 0,Y 72.674,Z 303.878,A -85,B 0,C 180,E1 -30809.503,E2 -30809.503} C_VEL
LIN {X 0,Y 67.214,Z 315.873,A -85,B 0,C 180,E1 -30811.114,E2 -30811.114} C_VEL
LIN {X 0,Y 60.93,Z 326.786,A -85,B 0,C 180,E1 -30813.255,E2 -30813.255} C_VEL
LIN {X 0,Y 53.521,Z 337.322,A -85,B 0,C 180,E1 -30816.461,E2 -30816.461} C_VEL
LIN {X 0,Y 45.94,Z 346.264,A -85,B 0,C 180,E1 -30820.783,E2 -30820.783} C_VEL
LIN {X 0,Y 41.794,Z 350.267,A -85,B 0,C 180,E1 -30822.773,E2 -30822.773} C_VEL
LIN {X 0,Y 30.728,Z 358.5,A -85,B 0,C 180,E1 -30825.581,E2 -30825.581} C_VEL
LIN {X 0,Y 24.318,Z 362.753,A -85,B 0,C 180,E1 -30829.648,E2 -30829.648} C_VEL
LIN {X 0,Y 21.453,Z 364.765,A -85,B 0,C 180,E1 -30834.203,E2 -30834.203} C_VEL
LIN {X 0,Y 14.148,Z 370.631,A -85,B 0,C 180,E1 -30863.4,E2 -30863.4} C_VEL
LIN {X 0,Y 14.322,Z 375.626,A -85,B 0,C 180,E1 -30917.407,E2 -30917.407} C_VEL
LIN {X 0,Y 21.819,Z 378.731,A -85,B 0,C 180,E1 -30945.101,E2 -30945.101} C_VEL
LIN {X 0,Y 28.25,Z 380.202,A -85,B 0,C 180,E1 -30954.361,E2 -30954.361} C_VEL
LIN {X 0,Y 35.141,Z 381.246,A -85,B 0,C 180,E1 -30960.194,E2 -30960.194} C_VEL
LIN {X 0,Y 42.281,Z 381.813,A -85,B 0,C 180,E1 -30964.172,E2 -30964.172} C_VEL
LIN {X 0,Y 51.882,Z 381.9,A -85,B 0,C 180,E1 -30967.787,E2 -30967.787} C_VEL
LIN {X 0,Y 49.845,Z 382.009,A -85,B 0,C 180,E1 -30969.247,E2 -30969.247} C_VEL
LIN {X 0,Y 36.397,Z 381.813,A -85,B 0,C 180,E1 -30975.094,E2 -30975.094} C_VEL
LIN {X 0,Y 29.92,Z 381.155,A -85,B 0,C 180,E1 -30980.015,E2 -30980.015} C_VEL
LIN {X 0,Y 18.538,Z 378.658,A -85,B 0,C 180,E1 -31000.687,E2 -31000.687} C_VEL
LIN {X 0,Y 13.824,Z 375.732,A -85,B 0,C 180,E1 -31035.268,E2 -31035.268} C_VEL
LIN {X 0,Y 13.41,Z 374.522,A -85,B 0,C 180,E1 -31049.994,E2 -31049.994} C_VEL
LIN {X 0,Y 16.18,Z 369.927,A -85,B 0,C 180,E1 -31090.652,E2 -31090.652} C_VEL
LIN {X 0,Y 25.204,Z 362.902,A -85,B 0,C 180,E1 -31114.986,E2 -31114.986} C_VEL
LIN {X 0,Y 34.594,Z 355.246,A -85,B 0,C 180,E1 -31124.787,E2 -31124.787} C_VEL
LIN {X 0,Y 42.883,Z 347.406,A -85,B 0,C 180,E1 -31129.516,E2 -31129.516} C_VEL
LIN {X 0,Y 50.528,Z 338.909,A -85,B 0,C 180,E1 -31132.303,E2 -31132.303} C_VEL
LIN {X 0,Y 58.241,Z 328.43,A -85,B 0,C 180,E1 -31134.575,E2 -31134.575} C_VEL
LIN {X 0,Y 65.172,Z 316.871,A -85,B 0,C 180,E1 -31135.931,E2 -31135.931} C_VEL
LIN {X 0,Y 71.053,Z 304.096,A -85,B 0,C 180,E1 -31136.923,E2 -31136.923} C_VEL
LIN {X 0,Y 75.513,Z 290.763,A -85,B 0,C 180,E1 -31137.574,E2 -31137.574} C_VEL
LIN {X 0,Y 78.213,Z 278.794,A -85,B 0,C 180,E1 -31137.943,E2 -31137.943} C_VEL
LIN {X 0,Y 80.423,Z 261.664,A -85,B 0,C 180,E1 -31138.588,E2 -31138.588} C_VEL
LIN {X 0,Y 79.756,Z 257.862,A -85,B 0,C 180,E1 -31143.889,E2 -31143.889} C_VEL
LIN {X 0,Y 79.648,Z 256.765,A -85,B 0,C 180,E1 -31145.829,E2 -31145.829} C_VEL
LIN {X 0,Y 79.439,Z 256.718,A -85,B 0,C 180,E1 -31150.936,E2 -31150.936} C_VEL
LIN {X 0,Y 79.599,Z 257.583,A -85,B 0,C 180,E1 -31155.359,E2 -31155.359} C_VEL
LIN {X 0,Y 80.076,Z 260.22,A -85,B 0,C 180,E1 -31160.1,E2 -31160.1} C_VEL
LIN {X 0,Y 80.363,Z 261.667,A -85,B 0,C 180,E1 -31161.957,E2 -31161.957} C_VEL
LIN {X 0,Y 79.994,Z 265.001,A -85,B 0,C 180,E1 -31162.192,E2 -31162.192} C_VEL
LIN {X 0,Y 77.595,Z 281.055,A -85,B 0,C 180,E1 -31162.614,E2 -31162.614} C_VEL
LIN {X 0,Y 74.194,Z 294.312,A -85,B 0,C 180,E1 -31163.308,E2 -31163.308} C_VEL
LIN {X 0,Y 69.951,Z 305.85,A -85,B 0,C 180,E1 -31164.181,E2 -31164.181} C_VEL
LIN {X 0,Y 64.063,Z 318.014,A -85,B 0,C 180,E1 -31165.501,E2 -31165.501} C_VEL
LIN {X 0,Y 57.291,Z 328.991,A -85,B 0,C 180,E1 -31167.208,E2 -31167.208} C_VEL
LIN {X 0,Y 49.56,Z 339.107,A -85,B 0,C 180,E1 -31169.71,E2 -31169.71} C_VEL
LIN {X 0,Y 40.234,Z 349.138,A -85,B 0,C 180,E1 -31173.933,E2 -31173.933} C_VEL
LIN {X 0,Y 31.986,Z 356.574,A -85,B 0,C 180,E1 -31179.728,E2 -31179.728} C_VEL
LIN {X 0,Y 22.669,Z 363.864,A -85,B 0,C 180,E1 -31191.685,E2 -31191.685} C_VEL
LIN {X 0,Y 21.453,Z 364.765,A -85,B 0,C 180,E1 -31194.203,E2 -31194.203} C_VEL
LIN {X 0,Y 18.694,Z 366.687,A -85,B 0,C 180,E1 -31200.055,E2 -31200.055} C_VEL
LIN {X 0,Y 14.24,Z 369.313,A -85,B 0,C 180,E1 -31210.242,E2 -31210.242} C_VEL
LIN {X 0,Y 7.488,Z 374.399,A -85,B 0,C 180,E1 -31275.592,E2 -31275.592} C_VEL
LIN {X 0,Y 10.464,Z 376.271,A -85,B 0,C 180,E1 -31307.273,E2 -31307.273} C_VEL
LIN {X 0,Y 12.058,Z 376.841,A -85,B 0,C 180,E1 -31312.575,E2 -31312.575} C_VEL
LIN {X 0,Y 23.777,Z 379.933,A -85,B 0,C 180,E1 -31327.334,E2 -31327.334} C_VEL
LIN {X 0,Y 21.467,Z 379.522,A -85,B 0,C 180,E1 -31330.826,E2 -31330.826} C_VEL
LIN {X 0,Y 9.177,Z 376.134,A -85,B 0,C 180,E1 -31360.008,E2 -31360.008} C_VEL
LIN {X 0,Y 6.326,Z 373.715,A -85,B 0,C 180,E1 -31409.988,E2 -31409.988} C_VEL
LIN {X 0,Y 11.734,Z 368.98,A -85,B 0,C 180,E1 -31473.934,E2 -31473.934} C_VEL
LIN {X 0,Y 21.413,Z 362.934,A -85,B 0,C 180,E1 -31489.921,E2 -31489.921} C_VEL
LIN {X 0,Y 31.701,Z 355.359,A -85,B 0,C 180,E1 -31496.031,E2 -31496.031} C_VEL
LIN {X 0,Y 40.42,Z 347.61,A -85,B 0,C 180,E1 -31498.726,E2 -31498.726} C_VEL
LIN {X 0,Y 49.195,Z 338.19,A -85,B 0,C 180,E1 -31500.298,E2 -31500.298} C_VEL
LIN {X 0,Y 57.122,Z 327.624,A -85,B 0,C 180,E1 -31501.529,E2 -31501.529} C_VEL
LIN {X 0,Y 64.174,Z 315.959,A -85,B 0,C 180,E1 -31502.144,E2 -31502.144} C_VEL
LIN {X 0,Y 69.911,Z 303.538,A -85,B 0,C 180,E1 -31502.6,E2 -31502.6} C_VEL
LIN {X 0,Y 74.381,Z 290.286,A -85,B 0,C 180,E1 -31502.929,E2 -31502.929} C_VEL
LIN {X 0,Y 77.24,Z 277.469,A -85,B 0,C 180,E1 -31503.134,E2 -31503.134} C_VEL
LIN {X 0,Y 78.795,Z 265.807,A -85,B 0,C 180,E1 -31503.492,E2 -31503.492} C_VEL
LIN {X 0,Y 78.65,Z 263.733,A -85,B 0,C 180,E1 -31506.997,E2 -31506.997} C_VEL
LIN {X 0,Y 78.532,Z 263.839,A -85,B 0,C 180,E1 -31511.135,E2 -31511.135} C_VEL
LIN {X 0,Y 78.611,Z 264.649,A -85,B 0,C 180,E1 -31514.568,E2 -31514.568} C_VEL
LIN {X 0,Y 78.751,Z 265.871,A -85,B 0,C 180,E1 -31516.991,E2 -31516.991} C_VEL
LIN {X 0,Y 76.93,Z 278.69,A -85,B 0,C 180,E1 -31517.371,E2 -31517.371} C_VEL
LIN {X 0,Y 73.793,Z 291.793,A -85,B 0,C 180,E1 -31517.755,E2 -31517.755} C_VEL
LIN {X 0,Y 69.42,Z 304.296,A -85,B 0,C 180,E1 -31518.354,E2 -31518.354} C_VEL
LIN {X 0,Y 64.097,Z 315.581,A -85,B 0,C 180,E1 -31519.016,E2 -31519.016} C_VEL
LIN {X 0,Y 57.027,Z 327.287,A -85,B 0,C 180,E1 -31520.001,E2 -31520.001} C_VEL
LIN {X 0,Y 49.054,Z 337.857,A -85,B 0,C 180,E1 -31521.371,E2 -31521.371} C_VEL
LIN {X 0,Y 40.197,Z 347.325,A -85,B 0,C 180,E1 -31523.384,E2 -31523.384} C_VEL
LIN {X 0,Y 29.646,Z 356.514,A -85,B 0,C 180,E1 -31527.258,E2 -31527.258} C_VEL
LIN {X 0,Y 19.224,Z 363.899,A -85,B 0,C 180,E1 -31534.662,E2 -31534.662} C_VEL
LIN {X 0,Y 9.199,Z 369.934,A -85,B 0,C 180,E1 -31557.051,E2 -31557.051} C_VEL
LIN {X 0,Y 7.821,Z 375.156,A -85,B 0,C 180,E1 -31654.003,E2 -31654.003} C_VEL
LIN {X 0,Y 12.058,Z 376.841,A -85,B 0,C 180,E1 -31672.575,E2 -31672.575} C_VEL
LIN {X 0,Y 10.971,Z 376.627,A -85,B 0,C 180,E1 -31675.501,E2 -31675.501} C_VEL
LIN {X 0,Y 4.587,Z 374.658,A -85,B 0,C 180,E1 -31672.313,E2 -31672.313} C_VEL
LIN {X 0,Y 4.023,Z 371.3,A -85,B 0,C 180,E1 -31524.262,E2 -31524.262} C_VEL
LIN {X 0,Y 10.441,Z 368.163,A -85,B 0,C 180,E1 -31514.727,E2 -31514.727} C_VEL
LIN {X 0,Y 16.767,Z 364.657,A -85,B 0,C 180,E1 -31513.254,E2 -31513.254} C_VEL
LIN {X 0,Y 22.887,Z 360.777,A -85,B 0,C 180,E1 -31513.38,E2 -31513.38} C_VEL
LIN {X 0,Y 33.195,Z 353.01,A -85,B 0,C 180,E1 -31513.355,E2 -31513.355} C_VEL
LIN {X 0,Y 43.312,Z 343.56,A -85,B 0,C 180,E1 -31513.207,E2 -31513.207} C_VEL
LIN {X 0,Y 52.291,Z 333.11,A -85,B 0,C 180,E1 -31512.997,E2 -31512.997} C_VEL
LIN {X 0,Y 60.346,Z 321.283,A -85,B 0,C 180,E1 -31512.748,E2 -31512.748} C_VEL
LIN {X 0,Y 66.331,Z 310.152,A -85,B 0,C 180,E1 -31512.551,E2 -31512.551} C_VEL
LIN {X 0,Y 71.466,Z 297.543,A -85,B 0,C 180,E1 -31512.375,E2 -31512.375} C_VEL
LIN {X 0,Y 75.301,Z 284.245,A -85,B 0,C 180,E1 -31512.1,E2 -31512.1} C_VEL
LIN {X 0,Y 77.574,Z 271.506,A -85,B 0,C 180,E1 -31512.036,E2 -31512.036} C_VEL
LIN {X 0,Y 77.625,Z 271.043,A -85,B 0,C 180,E1 -31511.735,E2 -31511.735} C_VEL
LIN {X 0,Y 77.668,Z 270.732,A -85,B 0,C 180,E1 -31508.512,E2 -31508.512} C_VEL
LIN {X 0,Y 75.313,Z 284.29,A -85,B 0,C 180,E1 -31508.357,E2 -31508.357} C_VEL
LIN {X 0,Y 71.393,Z 297.848,A -85,B 0,C 180,E1 -31508.426,E2 -31508.426} C_VEL
LIN {X 0,Y 66.61,Z 309.659,A -85,B 0,C 180,E1 -31508.452,E2 -31508.452} C_VEL
LIN {X 0,Y 60.411,Z 321.275,A -85,B 0,C 180,E1 -31508.571,E2 -31508.571} C_VEL
LIN {X 0,Y 53.305,Z 331.844,A -85,B 0,C 180,E1 -31508.579,E2 -31508.579} C_VEL
LIN {X 0,Y 45.507,Z 341.293,A -85,B 0,C 180,E1 -31508.585,E2 -31508.585} C_VEL
LIN {X 0,Y 35.578,Z 351.048,A -85,B 0,C 180,E1 -31509.011,E2 -31509.011} C_VEL
LIN {X 0,Y 24.897,Z 359.436,A -85,B 0,C 180,E1 -31508.907,E2 -31508.907} C_VEL
LIN {X 0,Y 14.262,Z 366.131,A -85,B 0,C 180,E1 -31509.792,E2 -31509.792} C_VEL
LIN {X 0,Y 14.383,Z 366.041,A -85,B 0,C 180,E1 -31512.268,E2 -31512.268} C_VEL
LIN {X 0,Y 22.887,Z 360.777,A -85,B 0,C 180,E1 -31513.38,E2 -31513.38} C_VEL
LIN {X 0,Y 25.995,Z 362.44,A -85,B 0,C 180,E1 -31513.636,E2 -31513.636} C_VEL
LIN {X 0,Y 25.995,Z 600,A -85,B 0,C 180,E1 -31513.636,E2 -31513.636} C_VEL
LIN {X 0,Y 25.995,Z 600,A -85,B 0,C 180,E1 -31513.636,E2 -31513.636}

QRS_NEXT_CUT()

QRS_NEXT()
QRS_HOME()

END
